// TIA Portal project "ABB_umrichter_Profinet" (V14)

(* hardware
DEVICE "S7-1200-Station_1"  S7-1200 Station
   slot 0: "Baugruppenträger_0"  S7-1200 Rack  Rack  V1.0
   slot 1: "PLC_1"  CPU 1214C DC/DC/DC  6ES7 214-1AG40-0XB0  V4.2
DEVICE "GSD-Geraet_1"  GSD.Device.PN
   slot 0: "Baugruppenträger"  Rack  V1.0
   slot 0: "FENA"  FENA-11  6438177287445  V3.2.0
      slot 0: "FENA-11"  FENA-11
      slot 1: "Interface"  Interface
         slot 1: "Port 1"  Port 1
   slot 1: "PPO Type 6_1"  PPO Type 6  V3.2.0
      slot 0: "PPO6 Data Object"  PPO6 Data Object
*)

// ===== PLC "PLC_1"  CPU 1214C DC/DC/DC =====

// folder: ABB_Datentypen

TYPE "ABB"
TITLE = ABB DRIVE CONTROL INPUT AND OUT FALGS
VERSION : 0.1
// Know_How_Protect
   STRUCT
      PPO_TYPE : "PPO_TYPE";
      ADAPTER_TYPE : "ADAPTER_TYPE";
      DRIVER_TYPE : "DRIVER_TYPE";
      DPV_MODE : "DPV_MODE";   // FALSE = DP-V0 ; TRUE = DP-V1
      SWITCH_ON : Bool;   // TRUE = switch on(power on);FALSE = switch off; start power on state machine
      START : Bool;   // TRUE = start enable modulation; FALSE = stop along currently activ stop ramp
      EMCY_STOP : Bool;   // Low active; emergency stop to drive: FALSE = stop by ramp TRUE = no stop
      COAST_STOP : Bool;   // TRUE = coast stop FALSE = normal operation eneble
      EXT_CTRL : Bool;   // External control place 2 EXT2
      RESET : Bool;   // Fault acknowled
      SPEED_REF : Int;   // Speed reference value: -20000...20000
      DONE : Bool;   // Execution finished when output DONE=TRUE
      ERR : Bool;   // Error occured during execution when output ERR=TRUE
      STOPPED : Bool;   // Drive stopped, not ready 0=ready
      RUNNING : Bool;   // Drive is modulating - following reference
      FAULT : Bool;   // Drive has a fault
      WARN : Bool;   // Drive has a warning
      EXT_RUN_ENABLE : Bool;   // External run enable singal received -> must be set to run
      LOACAL_CONTROL : Bool;   // Drive control location LOCAL
      EXT_CTRL_LOC : Bool;   // External control location EXT2 selected
      ERNO : Int;   // ErrorCode; see online help SFC14 or SFC15
      ACT_SPEED : Int;   // Speed actual value: -20000...20000
      MSW : Word;   // Main Status Word
      MCW : Word;   // Actual Main Control Word
      PARA_READ : Bool;   // Read parameter value
      PARA_WRITE : Bool;   // Write parameter value
      PARA_NUM : DInt;   // Parameter number: 3 digits = group, 2 digits = index; e.g Par 20.06 = 2006
      PARA_VALUE_IN : DInt;   // Write parameter value
      PARA_DONE : Bool;   // Pulse execution finished
      PARA_ERR : Bool;   // Error occured
      PARA_BUSY : Bool;   // Function block busy
      PARA_ERNO : Word;   // Error ID see FPBA or RBPA manual
      PARA_NUM_OUT : DInt;   // Parameter number: 3 digits = group, 2 digits = index; e.g Par 20.06 = 2006
      PARA_VALUE_OUT : DInt;   // Readed parameter value
      PZD3_OUT : Int;   // Write PZD3 value to drive
      PZD4_OUT : Int;   // Write PZD4 value to drive
      PZD5_OUT : Int;   // Write PZD5 value to drive
      PZD6_OUT : Int;   // Write PZD6 value to drive
      PZD7_OUT : Int;   // Write PZD7 value to drive
      PZD8_OUT : Int;   // Write PZD8 value to drive
      PZD9_OUT : Int;   // Write PZD9 value to drive
      PZD10_OUT : Int;   // Write PZD10 value to drive
      PZD2_SCALED : Real;   // PZD2 scaled value
      PZD3_SCALED : Real;   // PZD3 scaled value
      PZD4_SCALED : Real;   // PZD4 scaled value
      PZD5_SCALED : Real;   // PZD5 scaled value
      PZD6_SCALED : Real;   // PZD6 scaled value
      PZD7_SCALED : Real;   // PZD7 scaled value
      PZD8_SCALED : Real;   // PZD8 scaled value
      PZD9_SCALED : Real;   // PZD9 scaled value
      PZD10_SCALED : Real;   // PZD10 scaled value
   END_STRUCT;
END_TYPE

// folder: ABB_Datentypen/SUBTYPE

TYPE "PPO_TYPE"
   STRUCT
      PPP_TYPE1 : Int := 1;
      PPP_TYPE2 : Int := 2;
      PPP_TYPE3 : Int := 3;
      PPP_TYPE4 : Int := 4;
      PPP_TYPE5 : Int := 5;
      PPP_TYPE6 : Int := 6;
      PPP_TYPE7 : Int := 7;
   END_STRUCT;
END_TYPE

TYPE "DRIVER_TYPE"
   STRUCT
      ACS800 : Int := 1;
      ACSM1 : Int := 2;
      ACS350 : Int := 3;
      ACS355 : Int := 4;
      ACS550 : Int := 5;
      ACS850 : Int := 6;
      ACS880 : Int := 7;
      ACS580 : Int := 8;
      ACS380 : Int := 9;
   END_STRUCT;
END_TYPE

TYPE "ADAPTER_TYPE"
   STRUCT
      "FPBA/FENA" : Int := 1;
      "RPBA/RETA" : Int := 2;
   END_STRUCT;
END_TYPE

TYPE "DPV_MODE"
   STRUCT
      DP_V0 : Bool;
      "DP_V1/Profinet" : Bool := true;
   END_STRUCT;
END_TYPE

// folder: (top level)

DATA_BLOCK "GVL"   // DB2
{ S7_Optimized_Access := 'TRUE' }
VERSION : 0.1
   VAR
      Drive_Param : "ABB";
   END_VAR
BEGIN
   // Drive_Param.SWITCH_ON : FALSE=Drive control switched off, TRUE=Drive control switched on. After an EMERGENCY STOP a new rising edge of SWITCH_ON is needed before next start. SWITCH_ON also needs to be active (TRUE) for resetting drive faults.
   // Drive_Param.START : FALSE=Ramp stop with deceleration time according to drive parameter, TRUE=Start. Drive start via fieldbus requires parameter setting in the drive.
   // Drive_Param.EMCY_STOP : FALSE=Emergency stop according to emergency stop deceleration time set in drive parameter, TRUE=Normal operation.
   // Drive_Param.COAST_STOP : FALSE=Normal operation, TRUE=Coast stop (drive releases control of the motor).
   // Drive_Param.EXT_CTRL : Selection of external control location EXT2. FALSE=EXT1, TRUE=EXT2. Shifting to EXT2 via fieldbus requires parameter setting in the drive.
   // Drive_Param.DPV_MODE : FALSE=DP-V01, TRUE=DP-V12 (or PROFINET).
   // Drive_Param.RESET : FALSE=No operation, TRUE =Reset drive fault.
   // Drive_Param.SPEED_REF : Speed reference value: -20000 to 20000. See chapter “Drive configuration” for scaling. Setting speed reference via fieldbus requires parameter setting in the drive.
   // Drive_Param.DONE : FALSE=Block execution not finished, TRUE=Block execution finished.
   // Drive_Param.ERR : FALSE=No error, TRUE=Error occurred during block execution.
   // Drive_Param.STOPPED : FALSE=Drive is not stopped, TRUE=Drive is stopped.
   // Drive_Param.RUNNING : FALSE=Drive is not running, TRUE=Drive is running and following the speed reference value.
   // Drive_Param.FAULT : FALSE=No drive fault active, TRUE=Drive fault active.
   // Drive_Param.WARN : FALSE=No drive warning active, TRUE=Drive warning active.FALSE=No drive warning active, TRUE=Drive warning active.
   // Drive_Param.EXT_RUN_ENABLE : FALSE=No external run enable signal received in the drive, TRUE=External run enable signal received in the drive.
   // Drive_Param.LOACAL_CONTROL : FALSE=Remote control (normal mode), TRUE=Local control (e.g. drive control panel or pc tool in local mode)
   // Drive_Param.EXT_CTRL_LOC : Actual control place, FALSE=EXT1, TRUE=EXT2.
   // Drive_Param.ERNO : Error code when ERR=TRUE, see SIMATIC online help for SFC14 or SFC15.
   // Drive_Param.ACT_SPEED : Drive actual speed: -20000 to 20000. See chapter “Drive configuration” for scaling.
   // Drive_Param.MSW : Drive main status word. See actual fieldbus adapter manual for detailed description.
   // Drive_Param.MCW : Drive main control word. See actual fieldbus adapter manual for detailed description.
   // Drive_Param.PARA_READ : Read the parameter value 0 -> 1 (executed on positive edge).
   // Drive_Param.PARA_WRITE : Write the parameter value 0 -> 1 (executed on positive edge).
   // Drive_Param.PARA_NUM : Read/written parameter: 3 numbers = group, 2 numbers =
   // Drive_Param.PARA_VALUE_IN : Parameter value to be written.
   // Drive_Param.PARA_DONE : FALSE=Block execution not finished, TRUE=Block execution finished.
   // Drive_Param.PARA_ERR : FALSE=No error, TRUE=Error occurred during block execution.
   // Drive_Param.PARA_BUSY : FALSE=No operation active, TRUE=Operation active.
   // Drive_Param.PARA_ERNO : Error code when ERR=TRUE.
   // Drive_Param.PARA_NUM_OUT : Handled parameter number: 3 numbers = group, 2 numbers = index; for example, Par 20.06 = 2006.
   // Drive_Param.PARA_VALUE_OUT : Read parameter value.
   // Drive_Param.PZD3_OUT : Write PZD3 value to the drive
   // Drive_Param.PZD4_OUT : Write PZD4 value to the drive
   // Drive_Param.PZD5_OUT : Write PZD5 value to the drive
   // Drive_Param.PZD6_OUT : Write PZD6 value to the drive
   // Drive_Param.PZD7_OUT : Write PZD7 value to the drive
   // Drive_Param.PZD8_OUT : Write PZD8 value to the drive
   // Drive_Param.PZD9_OUT : Write PZD9 value to the drive
   // Drive_Param.PZD10_OUT : Write PZD10 value to the drive
   // Drive_Param.PZD2_SCALED : Read PZD2 (actual speed / ACT) value from the drive, the default
   // Drive_Param.PZD3_SCALED : Read PZD3 value from the drive, the default scaling value is 1 = no
   // Drive_Param.PZD4_SCALED : Read PZD4 value from the drive, the default scaling value is 1 = no
   // Drive_Param.PZD5_SCALED : Read PZD5 value from the drive, the default scaling value is 1 = no
   // Drive_Param.PZD6_SCALED : Read PZD6 value from the drive, the default scaling value is 1 = no
   // Drive_Param.PZD7_SCALED : Read PZD7 value from the drive, the default scaling value is 1 = no
   // Drive_Param.PZD8_SCALED : Read PZD8 value from the drive, the default scaling value is 1 = no
   // Drive_Param.PZD9_SCALED : Read PZD9 value from the drive, the default scaling value is 1 = no
   // Drive_Param.PZD10_SCALED : Read PZD10 value from the drive, the default scaling value is 1 = no
   // Drive_Param.PPO_TYPE : The PPO type. 1, 2, 3, 4, 5 or 6; 0 = not allowed.
   // Drive_Param.ADAPTER_TYPE : PROFIBUS module type: FPBA-01 PROFIBUS DP module connected in the drive. 1=FPBA (or FENA), 2=RPBA (or RETA).
   // Drive_Param.DRIVER_TYPE : Drive type: ACS800=1, ACSM1=2, ACS350=3, ACS355=4, ACS550=5, ACS850=6, ACS880=7, ACS580=8, ACS380=9.
END_DATA_BLOCK

// folder: ABB_Umrichter

DATA_BLOCK "ABB_Umrichter_DB"   // DB5
{ S7_Optimized_Access := 'TRUE' }
VERSION : 0.1
// stored: InstanceOfName ABB_Umrichter
"ABB_Umrichter"
BEGIN
END_DATA_BLOCK

// folder: ABB_Umrichter/DLL

DATA_BLOCK "ABB_DRIVE_CONTROL_DB"   // DB1
{ S7_Optimized_Access := 'FALSE' }
AUTHOR : ABB
FAMILY : DRIVES
NAME : ABB
VERSION : 1.2
// stored: InstanceOfName ABB_DRIVE_CONTROL
"ABB_DRIVE_CONTROL"
BEGIN
END_DATA_BLOCK

DATA_BLOCK "ACS_DRIVE_PARA_DB"   // DB3
{ S7_Optimized_Access := 'FALSE' }
AUTHOR : ABB
FAMILY : DRIVES
NAME : ABB
VERSION : 1.2
// stored: InstanceOfName ACS_DRIVE_PARA
"ACS_DRIVE_PARA"
BEGIN
END_DATA_BLOCK

DATA_BLOCK "ACS_DRIVE_PZD_DB"   // DB4
{ S7_Optimized_Access := 'FALSE' }
AUTHOR : ABB
FAMILY : DRIVES
NAME : ABB
VERSION : 1.2
// stored: InstanceOfName ACS_DRIVE_PZD
"ACS_DRIVE_PZD"
BEGIN
END_DATA_BLOCK

// folder: (top level)

ORGANIZATION_BLOCK "Main"   // OB1, LAD, ProgramCycle
TITLE = "Main Program Sweep (Cycle)"
{ S7_Optimized_Access := 'TRUE' }
VERSION : 0.1
   VAR_INPUT
      Initial_Call : Bool;   // Initial call of this OB
      Remanence : Bool;   // =True, if remanent data are available
   END_VAR
BEGIN

REGION Network 1
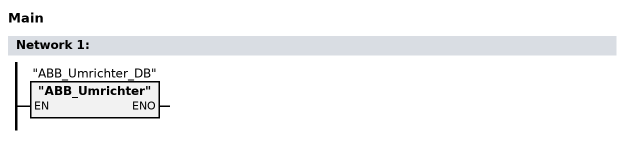
   RUNG wire#powerrail
      "ABB_Umrichter_DB"()
   END_RUNG
   // the same network as SCL:
   "ABB_Umrichter_DB"();   // "ABB_Umrichter"
END_REGION
END_ORGANIZATION_BLOCK

// folder: ABB_Umrichter

FUNCTION_BLOCK "ABB_Umrichter"   // FB1, LAD
{ S7_Optimized_Access := 'TRUE' }
VERSION : 0.1
BEGIN

REGION Network 1
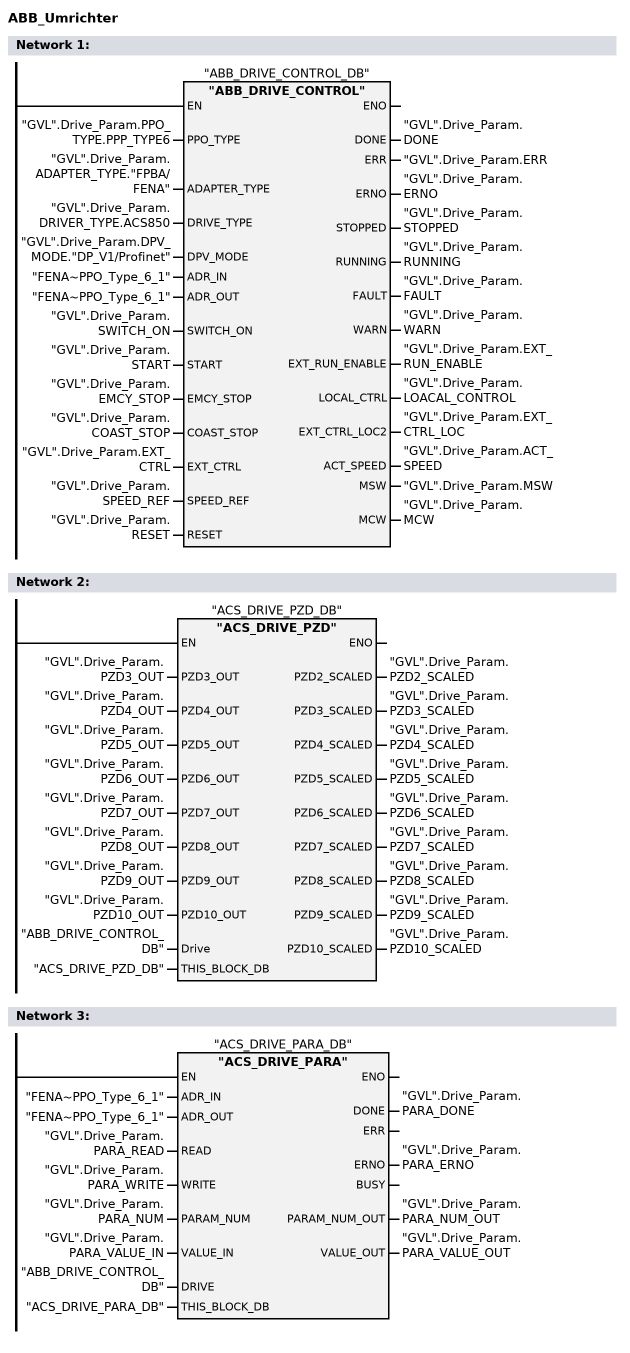
   RUNG wire#powerrail
      "ABB_DRIVE_CONTROL_DB"(PPO_TYPE := "GVL".Drive_Param.PPO_TYPE.PPP_TYPE6, ADAPTER_TYPE := "GVL".Drive_Param.ADAPTER_TYPE."FPBA/FENA", DRIVE_TYPE := "GVL".Drive_Param.DRIVER_TYPE.ACS850, DPV_MODE := "GVL".Drive_Param.DPV_MODE."DP_V1/Profinet", ADR_IN := "FENA~PPO_Type_6_1", ADR_OUT := "FENA~PPO_Type_6_1", SWITCH_ON := "GVL".Drive_Param.SWITCH_ON, START := "GVL".Drive_Param.START, EMCY_STOP := "GVL".Drive_Param.EMCY_STOP, COAST_STOP := "GVL".Drive_Param.COAST_STOP, EXT_CTRL := "GVL".Drive_Param.EXT_CTRL, SPEED_REF := "GVL".Drive_Param.SPEED_REF, RESET := "GVL".Drive_Param.RESET, DONE => "GVL".Drive_Param.DONE, ERR => "GVL".Drive_Param.ERR, ERNO => "GVL".Drive_Param.ERNO, STOPPED => "GVL".Drive_Param.STOPPED, RUNNING => "GVL".Drive_Param.RUNNING, FAULT => "GVL".Drive_Param.FAULT, WARN => "GVL".Drive_Param.WARN, EXT_RUN_ENABLE => "GVL".Drive_Param.EXT_RUN_ENABLE, LOCAL_CTRL => "GVL".Drive_Param.LOACAL_CONTROL, EXT_CTRL_LOC2 => "GVL".Drive_Param.EXT_CTRL_LOC, ACT_SPEED => "GVL".Drive_Param.ACT_SPEED, MSW => "GVL".Drive_Param.MSW, MCW => "GVL".Drive_Param.MCW)
   END_RUNG
   // the same network as SCL:
   "ABB_DRIVE_CONTROL_DB"(PPO_TYPE := "GVL".Drive_Param.PPO_TYPE.PPP_TYPE6,   // "ABB_DRIVE_CONTROL"
                          ADAPTER_TYPE := "GVL".Drive_Param.ADAPTER_TYPE."FPBA/FENA",
                          DRIVE_TYPE := "GVL".Drive_Param.DRIVER_TYPE.ACS850,
                          DPV_MODE := "GVL".Drive_Param.DPV_MODE."DP_V1/Profinet",
                          ADR_IN := "FENA~PPO_Type_6_1",
                          ADR_OUT := "FENA~PPO_Type_6_1",
                          SWITCH_ON := "GVL".Drive_Param.SWITCH_ON,
                          START := "GVL".Drive_Param.START,
                          EMCY_STOP := "GVL".Drive_Param.EMCY_STOP,
                          COAST_STOP := "GVL".Drive_Param.COAST_STOP,
                          EXT_CTRL := "GVL".Drive_Param.EXT_CTRL,
                          SPEED_REF := "GVL".Drive_Param.SPEED_REF,
                          RESET := "GVL".Drive_Param.RESET,
                          DONE => "GVL".Drive_Param.DONE,
                          ERR => "GVL".Drive_Param.ERR,
                          ERNO => "GVL".Drive_Param.ERNO,
                          STOPPED => "GVL".Drive_Param.STOPPED,
                          RUNNING => "GVL".Drive_Param.RUNNING,
                          FAULT => "GVL".Drive_Param.FAULT,
                          WARN => "GVL".Drive_Param.WARN,
                          EXT_RUN_ENABLE => "GVL".Drive_Param.EXT_RUN_ENABLE,
                          LOCAL_CTRL => "GVL".Drive_Param.LOACAL_CONTROL,
                          EXT_CTRL_LOC2 => "GVL".Drive_Param.EXT_CTRL_LOC,
                          ACT_SPEED => "GVL".Drive_Param.ACT_SPEED,
                          MSW => "GVL".Drive_Param.MSW,
                          MCW => "GVL".Drive_Param.MCW);
END_REGION

REGION Network 2
   RUNG wire#powerrail
      "ACS_DRIVE_PZD_DB"(PZD3_OUT := "GVL".Drive_Param.PZD3_OUT, PZD4_OUT := "GVL".Drive_Param.PZD4_OUT, PZD5_OUT := "GVL".Drive_Param.PZD5_OUT, PZD6_OUT := "GVL".Drive_Param.PZD6_OUT, PZD7_OUT := "GVL".Drive_Param.PZD7_OUT, PZD8_OUT := "GVL".Drive_Param.PZD8_OUT, PZD9_OUT := "GVL".Drive_Param.PZD9_OUT, PZD10_OUT := "GVL".Drive_Param.PZD10_OUT, Drive := "ABB_DRIVE_CONTROL_DB", THIS_BLOCK_DB := "ACS_DRIVE_PZD_DB", PZD2_SCALED => "GVL".Drive_Param.PZD2_SCALED, PZD3_SCALED => "GVL".Drive_Param.PZD3_SCALED, PZD4_SCALED => "GVL".Drive_Param.PZD4_SCALED, PZD5_SCALED => "GVL".Drive_Param.PZD5_SCALED, PZD6_SCALED => "GVL".Drive_Param.PZD6_SCALED, PZD7_SCALED => "GVL".Drive_Param.PZD7_SCALED, PZD8_SCALED => "GVL".Drive_Param.PZD8_SCALED, PZD9_SCALED => "GVL".Drive_Param.PZD9_SCALED, PZD10_SCALED => "GVL".Drive_Param.PZD10_SCALED)
   END_RUNG
   // the same network as SCL:
   "ACS_DRIVE_PZD_DB"(PZD3_OUT := "GVL".Drive_Param.PZD3_OUT,   // "ACS_DRIVE_PZD"
                      PZD4_OUT := "GVL".Drive_Param.PZD4_OUT,
                      PZD5_OUT := "GVL".Drive_Param.PZD5_OUT,
                      PZD6_OUT := "GVL".Drive_Param.PZD6_OUT,
                      PZD7_OUT := "GVL".Drive_Param.PZD7_OUT,
                      PZD8_OUT := "GVL".Drive_Param.PZD8_OUT,
                      PZD9_OUT := "GVL".Drive_Param.PZD9_OUT,
                      PZD10_OUT := "GVL".Drive_Param.PZD10_OUT,
                      Drive := "ABB_DRIVE_CONTROL_DB",
                      THIS_BLOCK_DB := "ACS_DRIVE_PZD_DB",
                      PZD2_SCALED => "GVL".Drive_Param.PZD2_SCALED,
                      PZD3_SCALED => "GVL".Drive_Param.PZD3_SCALED,
                      PZD4_SCALED => "GVL".Drive_Param.PZD4_SCALED,
                      PZD5_SCALED => "GVL".Drive_Param.PZD5_SCALED,
                      PZD6_SCALED => "GVL".Drive_Param.PZD6_SCALED,
                      PZD7_SCALED => "GVL".Drive_Param.PZD7_SCALED,
                      PZD8_SCALED => "GVL".Drive_Param.PZD8_SCALED,
                      PZD9_SCALED => "GVL".Drive_Param.PZD9_SCALED,
                      PZD10_SCALED => "GVL".Drive_Param.PZD10_SCALED);
END_REGION

REGION Network 3
   RUNG wire#powerrail
      "ACS_DRIVE_PARA_DB"(ADR_IN := "FENA~PPO_Type_6_1", ADR_OUT := "FENA~PPO_Type_6_1", READ := "GVL".Drive_Param.PARA_READ, WRITE := "GVL".Drive_Param.PARA_WRITE, PARAM_NUM := "GVL".Drive_Param.PARA_NUM, VALUE_IN := "GVL".Drive_Param.PARA_VALUE_IN, DRIVE := "ABB_DRIVE_CONTROL_DB", THIS_BLOCK_DB := "ACS_DRIVE_PARA_DB", DONE => "GVL".Drive_Param.PARA_DONE, ERR =>, ERNO => "GVL".Drive_Param.PARA_ERNO, BUSY =>, PARAM_NUM_OUT => "GVL".Drive_Param.PARA_NUM_OUT, VALUE_OUT => "GVL".Drive_Param.PARA_VALUE_OUT)
   END_RUNG
   // the same network as SCL:
   "ACS_DRIVE_PARA_DB"(ADR_IN := "FENA~PPO_Type_6_1",   // "ACS_DRIVE_PARA"
                       ADR_OUT := "FENA~PPO_Type_6_1",
                       READ := "GVL".Drive_Param.PARA_READ,
                       WRITE := "GVL".Drive_Param.PARA_WRITE,
                       PARAM_NUM := "GVL".Drive_Param.PARA_NUM,
                       VALUE_IN := "GVL".Drive_Param.PARA_VALUE_IN,
                       DRIVE := "ABB_DRIVE_CONTROL_DB",
                       THIS_BLOCK_DB := "ACS_DRIVE_PARA_DB",
                       DONE => "GVL".Drive_Param.PARA_DONE,
                       ERNO => "GVL".Drive_Param.PARA_ERNO,
                       PARAM_NUM_OUT => "GVL".Drive_Param.PARA_NUM_OUT,
                       VALUE_OUT => "GVL".Drive_Param.PARA_VALUE_OUT);
END_REGION
END_FUNCTION_BLOCK

// folder: ABB_Umrichter/DLL

FUNCTION_BLOCK "ABB_DRIVE_CONTROL"   // FB500, LAD
TITLE = ABB_DRIVE_CONTROL_FB
{ S7_Optimized_Access := 'FALSE' }
AUTHOR : ABB
FAMILY : DRIVES
NAME : ABB
VERSION : 1.2
   VAR_INPUT
      PPO_TYPE : Int;   // PPO-Type: 1,2,3,4,5 or 6; 0 = no fuction
      ADAPTER_TYPE : Int;   // AdapterType:FPBA=1,RPBA=2,FENA=3
      DRIVE_TYPE : Int;   // DriveType: ACS800=1,ACSM1=2,ACS350=3,ACS355=4,ACS550=5,ACS850=6,ACS880=7,ACS580=8,ACS380=9
      DPV_MODE : Bool;   // FALSE = DP-V0 ; TRUE = DP-V1
      ADR_IN : Hw_Io;   // Address of first input byte
      ADR_OUT : Hw_Io;   // Address of first output byte
      SWITCH_ON : Bool;   // TRUE = switch on(power on);FALSE = switch off; start power on state machine
      START : Bool;   // TRUE = start enable modulation; FALSE = stop along currently activ stop ramp
      EMCY_STOP : Bool;   // Low active; emergency stop to drive: FALSE = stop by ramp TRUE = no stop
      COAST_STOP : Bool;   // TRUE = coast stop FALSE = normal operation eneble
      EXT_CTRL : Bool;   // External control place 2 EXT2
      SPEED_REF : Int;   // Speed reference value: -20000...20000
   END_VAR
   VAR_OUTPUT
      DONE : Bool;   // Execution finished when output DONE=TRUE
      ERR : Bool;   // Error occured during execution when output ERR=TRUE
      ERNO : Int;   // ErrorCode; see online help SFC14 or SFC15
      STOPPED : Bool;   // The drive has been stopped
      RUNNING : Bool;   // Drive is modulating - following reference
      FAULT : Bool;   // Drive has a fault
      WARN : Bool;   // Drive has a warning
      EXT_RUN_ENABLE : Bool;   // External run enable singal received -> must be set to run
      LOCAL_CTRL : Bool;   // Drive control location LOCAL
      EXT_CTRL_LOC2 : Bool;   // External control location EXT2 selected
      ACT_SPEED : Int;   // Speed actual value: -20000...20000
      MSW : Word;   // Main Status Word
      MCW : Word;   // Actual Main Control Word
   END_VAR
   VAR_IN_OUT
      RESET : Bool;   // Fault acknowled
   END_VAR
   VAR
      Input : Struct
         PPO1 : Struct
            SW : Struct
               AT_SET_POINT : Bool;   // Speed within setpoints
               REMONTE : Bool;   // Profibus control allowed
               ABOVE_LIMIT : Bool;   // Speed / frequency across borders
               EXT_CTRL_LOC : Bool;   // 0=EXT1 1=EXT2 selected
               EXT_RUN_ENABLE : Bool;   // Injury Prevention
               MSV13 : Bool;   // Not in Use
               MSV14 : Bool;   // Not in Use
               COOM_FAULT : Bool;   // Communication Fault Profibus Module CH0
               RDY_ON : Bool;   // Startup finished
               RDY_RUN : Bool;   // Action Completed
               RDY_REF : Bool;   // In Progress
               TRIPPED : Bool;   // Interference
               OFF2_STATE : Bool;   // Freedom freely in the wheels
               OFF3_STATE : Bool;   // Stop as fast as possible
               ON_INHIB : Bool;   // Startup blocked
               ALARM : Bool;   // Alarm
            END_STRUCT;
            Act_Speed : Int;   // Speed
         END_STRUCT;
         PPO2 : Struct
            SW : Struct
               AT_SET_POINT : Bool;   // Speed within setpoints
               REMONTE : Bool;   // Profibus control allowed
               ABOVE_LIMIT : Bool;   // Speed / frequency across borders
               EXT_CTRL_LOC : Bool;   // 0=EXT1 1=EXT2 selected
               EXT_RUN_ENABLE : Bool;   // Injury Prevention
               MSV13 : Bool;   // Not in Use
               MSV14 : Bool;   // Not in Use
               COOM_FAULT : Bool;   // Communication Fault Profibus Module CH0
               RDY_ON : Bool;   // Startup finished
               RDY_RUN : Bool;   // Action Completed
               RDY_REF : Bool;   // In Progress
               TRIPPED : Bool;   // Interference
               OFF2_STATE : Bool;   // Freedom freely in the wheels
               OFF3_STATE : Bool;   // Stop as fast as possible
               ON_INHIB : Bool;   // Startup blocked
               ALARM : Bool;   // Alarm
            END_STRUCT;
            Act_Speed : Int;   // Speed
            PZD_3 : Int;
            PZD_4 : Int;
            PZD_5 : Int;
            PZD_6 : Int;
         END_STRUCT;
         PPO3 : Struct
            SW : Struct
               AT_SET_POINT : Bool;   // Speed within setpoints
               REMONTE : Bool;   // Profibus control allowed
               ABOVE_LIMIT : Bool;   // Speed / frequency across borders
               EXT_CTRL_LOC : Bool;   // 0=EXT1 1=EXT2 selected
               EXT_RUN_ENABLE : Bool;   // Injury Prevention
               MSV13 : Bool;   // Not in Use
               MSV14 : Bool;   // Not in Use
               COOM_FAULT : Bool;   // Communication Fault Profibus Module CH0
               RDY_ON : Bool;   // Startup finished
               RDY_RUN : Bool;   // Action Completed
               RDY_REF : Bool;   // In Progress
               TRIPPED : Bool;   // Interference
               OFF2_STATE : Bool;   // Freedom freely in the wheels
               OFF3_STATE : Bool;   // Stop as fast as possible
               ON_INHIB : Bool;   // Startup blocked
               ALARM : Bool;   // Alarm
            END_STRUCT;
            Act_Speed : Int;   // Speed
         END_STRUCT;
         PPO4 : Struct
            SW : Struct
               AT_SET_POINT : Bool;   // Speed within setpoints
               REMONTE : Bool;   // Profibus control allowed
               ABOVE_LIMIT : Bool;   // Speed / frequency across borders
               EXT_CTRL_LOC : Bool;   // 0=EXT1 1=EXT2 selected
               EXT_RUN_ENABLE : Bool;   // Injury Prevention
               MSV13 : Bool;   // Not in Use
               MSV14 : Bool;   // Not in Use
               COOM_FAULT : Bool;   // Communication Fault Profibus Module CH0
               RDY_ON : Bool;   // Startup finished
               RDY_RUN : Bool;   // Action Completed
               RDY_REF : Bool;   // In Progress
               TRIPPED : Bool;   // Interference
               OFF2_STATE : Bool;   // Freedom freely in the wheels
               OFF3_STATE : Bool;   // Stop as fast as possible
               ON_INHIB : Bool;   // Startup blocked
               ALARM : Bool;   // Alarm
            END_STRUCT;
            Act_Speed : Int;   // Speed
            PZD_3 : Int;
            PZD_4 : Int;
            PZD_5 : Int;
            PZD_6 : Int;
         END_STRUCT;
         PPO5 : Struct
            SW : Struct
               AT_SET_POINT : Bool;   // Speed within setpoints
               REMONTE : Bool;   // Profibus control allowed
               ABOVE_LIMIT : Bool;   // Speed / frequency across borders
               EXT_CTRL_LOC : Bool;   // 0=EXT1 1=EXT2 selected
               EXT_RUN_ENABLE : Bool;   // Injury Prevention
               MSV13 : Bool;   // Not in Use
               MSV14 : Bool;   // Not in Use
               COOM_FAULT : Bool;   // Communication Fault Profibus Module CH0
               RDY_ON : Bool;   // Startup finished
               RDY_RUN : Bool;   // Action Completed
               RDY_REF : Bool;   // In Progress
               TRIPPED : Bool;   // Interference
               OFF2_STATE : Bool;   // Freedom freely in the wheels
               OFF3_STATE : Bool;   // Stop as fast as possible
               ON_INHIB : Bool;   // Startup blocked
               ALARM : Bool;   // Alarm
            END_STRUCT;
            Act_Speed : Int;   // Speed
            PZD_3 : Int;
            PZD_4 : Int;
            PZD_5 : Int;
            PZD_6 : Int;
            PZD_7 : Int;
            PZD_8 : Int;
            PZD_9 : Int;
            PZD_10 : Int;
         END_STRUCT;
         PPO6 : Struct
            SW : Struct
               AT_SET_POINT : Bool;   // Speed within setpoints
               REMONTE : Bool;   // Profibus control allowed
               ABOVE_LIMIT : Bool;   // Speed / frequency across borders
               EXT_CTRL_LOC : Bool;   // 0=EXT1 1=EXT2 selected
               EXT_RUN_ENABLE : Bool;   // Injury Prevention
               MSV13 : Bool;   // Not in Use
               MSV14 : Bool;   // Not in Use
               COOM_FAULT : Bool;   // Communication Fault Profibus Module CH0
               RDY_ON : Bool;   // Startup finished
               RDY_RUN : Bool;   // Action Completed
               RDY_REF : Bool;   // In Progress
               TRIPPED : Bool;   // Interference
               OFF2_STATE : Bool;   // Freedom freely in the wheels
               OFF3_STATE : Bool;   // Stop as fast as possible
               ON_INHIB : Bool;   // Startup blocked
               ALARM : Bool;   // Alarm
            END_STRUCT;
            Act_Speed : Int;   // Speed
            PZD_3 : Int;
            PZD_4 : Int;
            PZD_5 : Int;
            PZD_6 : Int;
            PZD_7 : Int;
            PZD_8 : Int;
            PZD_9 : Int;
            PZD_10 : Int;
         END_STRUCT;
         ACT : Struct
            SW : Struct
               AT_SET_POINT : Bool;   // Speed within setpoints
               REMONTE : Bool;   // Profibus control allowed
               ABOVE_LIMIT : Bool;   // Speed / frequency across borders
               EXT_CTRL_LOC : Bool;   // 0=EXT1 1=EXT2 selected
               EXT_RUN_ENABLE : Bool;   // Injury Prevention
               MSV13 : Bool;   // Not in Use
               MSV14 : Bool;   // Not in Use
               COOM_FAULT : Bool;   // Communication Fault Profibus Module CH0
               RDY_ON : Bool;   // Startup finished
               RDY_RUN : Bool;   // Action Completed
               RDY_REF : Bool;   // In Progress
               TRIPPED : Bool;   // Interference
               OFF2_STATE : Bool;   // Freedom freely in the wheels
               OFF3_STATE : Bool;   // Stop as fast as possible
               ON_INHIB : Bool;   // Startup blocked
               ALARM : Bool;   // Alarm
            END_STRUCT;
            Act_Speed : Int;   // Speed
         END_STRUCT;
      END_STRUCT;
      Output : Struct
         PPO1 : Struct
            CW : Struct
               INCHING_1 : Bool;   // Standard Speed for instruction 1
               INCHING_2 : Bool;   // Standard Speed for instruction 2
               REMONTE_CMD : Bool;   // Profibus control for use
               EXT_CTRL_LOC : Bool;   // 0=EXT1 1=EXT2 selected
               RESERVE_2 : Bool;   // Not in Use
               RESERVE_3 : Bool;   // Not in Use
               RESERVE_4 : Bool;   // Not in Use
               RESERVE_5 : Bool;   // Not in Use
               OFF1 : Bool;   // Start up to readiness
               OFF2 : Bool;   // Free wheel stops
               OFF3 : Bool;   // Emergency stop stop
               INHIBIT_OPREATION : Bool;   // Go to control
               RAMP_OUT_ZERO : Bool;   // Control release
               RAMP_HOLD : Bool;   // Acceleration allowed
               RAMP_IN_ZERO : Bool;   // Speed instruction to zero
               RESET : Bool;   // Fault Reset
            END_STRUCT;
            RefSpeed : Int;
         END_STRUCT;
         PPO2 : Struct
            CW : Struct
               INCHING_1 : Bool;   // Standard Speed for instruction 1
               INCHING_2 : Bool;   // Standard Speed for instruction 2
               REMONTE_CMD : Bool;   // Profibus control for use
               EXT_CTRL_LOC : Bool;   // 0=EXT1 1=EXT2 selected
               RESERVE_2 : Bool;   // Not in Use
               RESERVE_3 : Bool;   // Not in Use
               RESERVE_4 : Bool;   // Not in Use
               RESERVE_5 : Bool;   // Not in Use
               OFF1 : Bool;   // Start up to readiness
               OFF2 : Bool;   // Free wheel stops
               OFF3 : Bool;   // Emergency stop stop
               INHIBIT_OPREATION : Bool;   // Go to control
               RAMP_OUT_ZERO : Bool;   // Control release
               RAMP_HOLD : Bool;   // Acceleration allowed
               RAMP_IN_ZERO : Bool;   // Speed instruction to zero
               RESET : Bool;   // Fault Reset
            END_STRUCT;
            RefSpeed : Int;
            PZD_3 : Int;
            PZD_4 : Int;
            PZD_5 : Int;
            PZD_6 : Int;
         END_STRUCT;
         PPO3 : Struct
            CW : Struct
               INCHING_1 : Bool;   // Standard Speed for instruction 1
               INCHING_2 : Bool;   // Standard Speed for instruction 2
               REMONTE_CMD : Bool;   // Profibus control for use
               EXT_CTRL_LOC : Bool;   // 0=EXT1 1=EXT2 selected
               RESERVE_2 : Bool;   // Not in Use
               RESERVE_3 : Bool;   // Not in Use
               RESERVE_4 : Bool;   // Not in Use
               RESERVE_5 : Bool;   // Not in Use
               OFF1 : Bool;   // Start up to readiness
               OFF2 : Bool;   // Free wheel stops
               OFF3 : Bool;   // Emergency stop stop
               INHIBIT_OPREATION : Bool;   // Go to control
               RAMP_OUT_ZERO : Bool;   // Control release
               RAMP_HOLD : Bool;   // Acceleration allowed
               RAMP_IN_ZERO : Bool;   // Speed instruction to zero
               RESET : Bool;   // Fault Reset
            END_STRUCT;
            RefSpeed : Int;
         END_STRUCT;
         PPO4 : Struct
            CW : Struct
               INCHING_1 : Bool;   // Standard Speed for instruction 1
               INCHING_2 : Bool;   // Standard Speed for instruction 2
               REMONTE_CMD : Bool;   // Profibus control for use
               EXT_CTRL_LOC : Bool;   // 0=EXT1 1=EXT2 selected
               RESERVE_2 : Bool;   // Not in Use
               RESERVE_3 : Bool;   // Not in Use
               RESERVE_4 : Bool;   // Not in Use
               RESERVE_5 : Bool;   // Not in Use
               OFF1 : Bool;   // Start up to readiness
               OFF2 : Bool;   // Free wheel stops
               OFF3 : Bool;   // Emergency stop stop
               INHIBIT_OPREATION : Bool;   // Go to control
               RAMP_OUT_ZERO : Bool;   // Control release
               RAMP_HOLD : Bool;   // Acceleration allowed
               RAMP_IN_ZERO : Bool;   // Speed instruction to zero
               RESET : Bool;   // Fault Reset
            END_STRUCT;
            RefSpeed : Int;
            PZD_3 : Int;
            PZD_4 : Int;
            PZD_5 : Int;
            PZD_6 : Int;
         END_STRUCT;
         PPO5 : Struct
            CW : Struct
               INCHING_1 : Bool;   // Standard Speed for instruction 1
               INCHING_2 : Bool;   // Standard Speed for instruction 2
               REMONTE_CMD : Bool;   // Profibus control for use
               EXT_CTRL_LOC : Bool;   // 0=EXT1 1=EXT2 selected
               RESERVE_2 : Bool;   // Not in Use
               RESERVE_3 : Bool;   // Not in Use
               RESERVE_4 : Bool;   // Not in Use
               RESERVE_5 : Bool;   // Not in Use
               OFF1 : Bool;   // Start up to readiness
               OFF2 : Bool;   // Free wheel stops
               OFF3 : Bool;   // Emergency stop stop
               INHIBIT_OPREATION : Bool;   // Go to control
               RAMP_OUT_ZERO : Bool;   // Control release
               RAMP_HOLD : Bool;   // Acceleration allowed
               RAMP_IN_ZERO : Bool;   // Speed instruction to zero
               RESET : Bool;   // Fault Reset
            END_STRUCT;
            RefSpeed : Int;
            PZD_3 : Int;
            PZD_4 : Int;
            PZD_5 : Int;
            PZD_6 : Int;
            PZD_7 : Int;
            PZD_8 : Int;
            PZD_9 : Int;
            PZD_10 : Int;
         END_STRUCT;
         PPO6 : Struct
            CW : Struct
               INCHING_1 : Bool;   // Standard Speed for instruction 1
               INCHING_2 : Bool;   // Standard Speed for instruction 2
               REMONTE_CMD : Bool;   // Profibus control for use
               EXT_CTRL_LOC : Bool;   // 0=EXT1 1=EXT2 selected
               RESERVE_2 : Bool;   // Not in Use
               RESERVE_3 : Bool;   // Not in Use
               RESERVE_4 : Bool;   // Not in Use
               RESERVE_5 : Bool;   // Not in Use
               OFF1 : Bool;   // Start up to readiness
               OFF2 : Bool;   // Free wheel stops
               OFF3 : Bool;   // Emergency stop stop
               INHIBIT_OPREATION : Bool;   // Go to control
               RAMP_OUT_ZERO : Bool;   // Control release
               RAMP_HOLD : Bool;   // Acceleration allowed
               RAMP_IN_ZERO : Bool;   // Speed instruction to zero
               RESET : Bool;   // Fault Reset
            END_STRUCT;
            RefSpeed : Int;
            PZD_3 : Int;
            PZD_4 : Int;
            PZD_5 : Int;
            PZD_6 : Int;
            PZD_7 : Int;
            PZD_8 : Int;
            PZD_9 : Int;
            PZD_10 : Int;
         END_STRUCT;
         ACT : Struct
            CW : Struct
               INCHING_1 : Bool;   // Standard Speed for instruction 1
               INCHING_2 : Bool;   // Standard Speed for instruction 2
               REMONTE_CMD : Bool;   // Profibus control for use
               EXT_CTRL_LOC : Bool;   // 0=EXT1 1=EXT2 selected
               RESERVE_2 : Bool;   // Not in Use
               RESERVE_3 : Bool;   // Not in Use
               RESERVE_4 : Bool;   // Not in Use
               RESERVE_5 : Bool;   // Not in Use
               OFF1 : Bool;   // Start up to readiness
               OFF2 : Bool;   // Free wheel stops
               OFF3 : Bool;   // Emergency stop stop
               INHIBIT_OPREATION : Bool;   // Go to control
               RAMP_OUT_ZERO : Bool;   // Control release
               RAMP_HOLD : Bool;   // Acceleration allowed
               RAMP_IN_ZERO : Bool;   // Speed instruction to zero
               RESET : Bool;   // Fault Reset
            END_STRUCT;
            RefSpeed : Int;
         END_STRUCT;
      END_STRUCT;
      PARA_INTERNAL_DPV0 : Struct
         Done : Bool;
         Err : Bool;
         Busy : Bool;
         Read_FB : Bool;
         Write_FB : Bool;
         Time_out : Bool;
         Read_request : Bool;
         Write_Request : Bool;
         Parameter_access : Bool;
         Para_9 : Bool;
         Para_10 : Bool;
         Para_11 : Bool;
         Para_12 : Bool;
         Para_13 : Bool;
         Para_14 : Bool;
         Para_15 : Bool;
         Para_16 : Bool;
         Para_17 : Bool;
         Para_18 : Bool;
         Para_19 : Bool;
         Para_20 : Bool;
         Para_21 : Bool;
         Para_22 : Bool;
         Para_23 : Bool;
         Para_24 : Bool;
         Para_25 : Bool;
         Para_26 : Bool;
         Para_27 : Bool;
         Para_28 : Bool;
         Para_29 : Bool;
         Para_30 : Bool;
         PDV_MODE : Bool;   // DP-V0 = 0 (false) / DP-V1 = 1 (true)
         RESPONCE_LABEL : Int;
         PARA_NUM_OUT : Int;
         PARA_NUM_INDEX_OUT : Int;
         PARA_ERR_NRO : Word;
         PARA_VALUE_OUT : DInt;
         ADDRESS_IN : Word;
         ADDRESS_OUT : Word;
         Master_to_Slave : Struct
            ID : Word;   // Request Label bits 4-7 Parameter number bits 0-2
            IND : Word;   // Parameter number index bits 0-15
            VALUE : DWord;   // Parameter values
         END_STRUCT;
         Slave_to_Master : Struct
            ID : Word;   // Request Label bits 4-7 Parameter number bits 0-2
            IND : Word;   // Parameter number index bits 0-15
            VALUE : DWord;   // Parameter values
         END_STRUCT;
         PPO_TYPE : Int;   // PPO-Type: 1,2,3,4,5 or 6; 0 = no fuction
         ADAPTER_TYPE : Int;   // AdapterType:FPBA=1,RPBA=2,FENA=3
         DRIVE_TYPE : Int;   // DiveType: ACS800=1,ACSM1=2,ACS350=3,ACS355=4,ACS550=5,ACS850=6,ACS880=7
      END_STRUCT;
      PARA_INTERNAL_DPV1 : Struct
         Request : Struct
            Reference : Byte;
            ID : Byte;   // 1 read / 2 change
            Axis : Byte;
            NoOfParameters : Byte;
            Attribute : Byte;
            NoOfElements : Byte;
            ParameterIndex : Word;
            Subindex : Word;
            Format : Byte;
            NumberOfValues : Byte;
            Value : DWord;
         END_STRUCT;
         Responce : Struct
            Reference : Byte;
            ID : Byte;
            Axis : Byte;
            NoOfParametrs : Byte;
            Format : Byte;
            NoOfValues : Byte;
            Value : DWord;
         END_STRUCT;
         Request_DONE : Bool;
         Request_BUSY : Bool;
         Request_ERROR : Bool;
         Request_STATUS : DWord;
         Responce_VALID : Bool;
         Responce_BUSY : Bool;
         Responce_ERROR : Bool;
         Responce_STATUS : DWord;
         Responce_LEN : UInt;
      END_STRUCT;
      INTERNAL_PZD : Struct
         IN : Struct
            PZD2 : Int;
            PZD3 : Int;
            PZD4 : Int;
            PZD5 : Int;
            PZD6 : Int;
            PZD7 : Int;
            PZD8 : Int;
            PZD9 : Int;
            PZD10 : Int;
         END_STRUCT;
         OUT : Struct
            PZD3 : Int;
            PZD4 : Int;
            PZD5 : Int;
            PZD6 : Int;
            PZD7 : Int;
            PZD8 : Int;
            PZD9 : Int;
            PZD10 : Int;
         END_STRUCT;
         SCALED : Struct
            PZD2 : Real;
            PZD3 : Real;
            PZD4 : Real;
            PZD5 : Real;
            PZD6 : Real;
            PZD7 : Real;
            PZD8 : Real;
            PZD9 : Real;
            PZD10 : Real;
         END_STRUCT;
         SCALE : Struct
            PZD2_SCALE : Real;
            PZD3_SCALE : Real;
            PZD4_SCALE : Real;
            PZD5_SCALE : Real;
            PZD6_SCALE : Real;
            PZD7_SCALE : Real;
            PZD8_SCALE : Real;
            PZD9_SCALE : Real;
            PZD10_SCALE : Real;
         END_STRUCT;
      END_STRUCT;
      DPV1_WRITE : WRREC;
      DPV1_READ : WRREC;
      DP1_RESPONCE : RDREC;
      INPUT_ADDRESS : Word;
      OUTPUT_ADDRESS : Word;
      RET_VAL_INPUT : Int;
      RET_VAL_OUTPUT : Int;
      DONE_ON : Bool;
      ParameterErr : Bool;
      ERROR : Bool;
      READ_FAULT : Bool;
      SWITCH_ON_FP : Bool;
      POWER_STATE : Int;
      ALLWAYS_ON : Bool;
      ALLWAYS_OFF : Bool;
      POWER_ON : Bool;
      RESET_POWER_ON : Bool;
      PARA_TIME_OUT : TON_TIME;
      INTERNA_ERR : Int;
      POWER_RESET_FB : Bool;
      PARA_NUM : DInt;
      PARA_VALUE : DInt;
      PARA_INTERNAL_DPV1_16bit : Struct
         Request : Struct
            Reference : Byte;
            ID : Byte;   // 1 read / 2 change
            Axis : Byte;
            NoOfParameters : Byte;
            Attribute : Byte := B#16#10;
            NoOfElements : Byte;
            ParameterIndex : Word;
            Subindex : Word;
            Format : Byte;
            NumberOfValues : Byte;
            Value : Word;
         END_STRUCT;
         Responce : Struct
            Reference : Byte;
            ID : Byte;
            Axis : Byte;
            NoOfParametrs : Byte;
            Format : Byte;
            NoOfValues : Byte;
            Value : DWord;
         END_STRUCT;
         Request_DONE : Bool;
         Request_BUSY : Bool;
         Request_ERROR : Bool;
         Request_STATUS : DWord;
         Responce_VALID : Bool;
         Responce_BUSY : Bool;
         Responce_ERROR : Bool;
         Responce_STATUS : DWord;
         Responce_LEN : Int;
      END_STRUCT;
      Drive_Type_Dummy : Bool;
      Drive_Type_Dummy2 : Bool;
      Response_Format_Dummy : Int;
      Format_Check : Bool;
      Format_Check_1 : Bool;
      Request_Sent_32bit : Bool;
      Request_Sent_16bit : Bool;
      Request_Sent_16bit_1 : Bool;
      RESTART : Bool;
      RESTART_EMG : Bool;
      POWER_RESET_FB_1 : Bool;
   END_VAR
   VAR_TEMP
      PARA_READ_ERR : Int;
      TEMP0 : Time;
      IN_ADDRESS_DW : Word;
      OUT_ADDRESS_DW : Word;
      dummy : Bool;
      MSW_Temp : Struct
         SW : Struct
            AT_SET_POINT : Bool;   // Nopeus asetusarvojen sisällä
            REMONTE : Bool;   // Profibuss ohjaus sallittu
            ABOVE_LIMIT : Bool;   // Nopeus / taajuus yli rajojen
            EXT_CTRL_LOC : Bool;   // 0=EXT1 1=EXT2 selected
            EXT_RUN_ENABLE : Bool;   // Vahinkokäynnistyksen esto
            MSV13 : Bool;   // Ei käytössä
            MSV14 : Bool;   // Ei käytössä
            COOM_FAULT : Bool;   // Kommunikointivika profibus moduuli CH0
            RDY_ON : Bool;   // Käynnistys valmis
            RDY_RUN : Bool;   // Toiminta valmis
            RDY_REF : Bool;   // Käynnissä
            TRIPPED : Bool;   // Häiriö
            OFF2_STATE : Bool;   // Pysäytys vapaasti pyörien
            OFF3_STATE : Bool;   // Pysäytys hahdollisimman nopeasti
            ON_INHIB : Bool;   // Käynnistys estetty
            ALARM : Bool;   // Hälytys
         END_STRUCT;
      END_STRUCT;
      MSW_Conv AT MSW_Temp : Word;
      MCW_Temp : Struct
         CW : Struct
            INCHING_1 : Bool;   // Vakio nopeus ohje 1 käyttöön
            INCHING_2 : Bool;   // Vakio nopeus ohje 2 käyttöön
            REMONTE_CMD : Bool;   // Profibuss ohjaus käyttöön
            EXT_CTRL_LOC : Bool;   // 0=EXT1 1=EXT2 selected
            RESERVE_2 : Bool;   // Ei käytössä
            RESERVE_3 : Bool;   // Ei käytössä
            RESERVE_4 : Bool;   // Ei käytössä
            RESERVE_5 : Bool;   // Ei käytössä
            OFF1 : Bool;   // Käynnistys valmiuteen
            OFF2 : Bool;   // Vapaastipyörien seis
            OFF3 : Bool;   // Hätä-seis pysäytys
            INHIBIT_OPREATION : Bool;   // Käyntiin ohjaus
            RAMP_OUT_ZERO : Bool;   // Ohjauksen vapautus
            RAMP_HOLD : Bool;   // Kiihdytys sallittu
            RAMP_IN_ZERO : Bool;   // Nopeus ohje nollaan
            RESET : Bool;   // Häiriön kuittaus
         END_STRUCT;
      END_STRUCT;
      MCW_Conv AT MCW_Temp : Word;
      "ReadRequest Sent" : Bool;
      PowerState_Temp : Int;
   END_VAR
   VAR_TEMP   // added for the SCL form of the ladder/FBD networks
      _w1 : Bool;
      _w2 : Bool;
      _w3 : Bool;
   END_VAR
BEGIN

REGION Network 1: Set init values
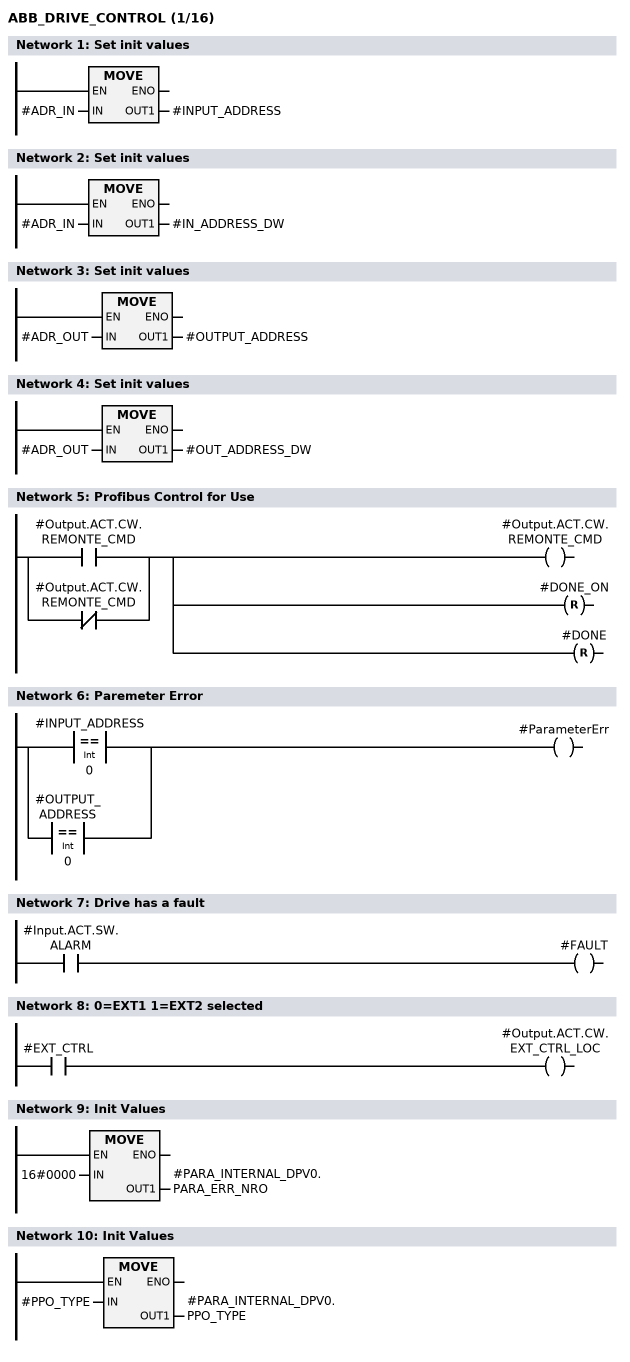
   RUNG wire#powerrail
      { S7_GenerateENO := "TRUE" } Move(in := #ADR_IN, out1 => #INPUT_ADDRESS)
   END_RUNG
   // the same network as SCL:
   #INPUT_ADDRESS := #ADR_IN;
END_REGION

REGION Network 2: Set init values
   RUNG wire#powerrail
      { S7_GenerateENO := "TRUE" } Move(in := #ADR_IN, out1 => #IN_ADDRESS_DW)
   END_RUNG
   // the same network as SCL:
   #IN_ADDRESS_DW := #ADR_IN;
END_REGION

REGION Network 3: Set init values
   RUNG wire#powerrail
      { S7_GenerateENO := "TRUE" } Move(in := #ADR_OUT, out1 => #OUTPUT_ADDRESS)
   END_RUNG
   // the same network as SCL:
   #OUTPUT_ADDRESS := #ADR_OUT;
END_REGION

REGION Network 4: Set init values
   RUNG wire#powerrail
      { S7_GenerateENO := "TRUE" } Move(in := #ADR_OUT, out1 => #OUT_ADDRESS_DW)
   END_RUNG
   // the same network as SCL:
   #OUT_ADDRESS_DW := #ADR_OUT;
END_REGION

REGION Network 5: Profibus Control for Use
   RUNG wire#powerrail
      Contact( #Output.ACT.CW.REMONTE_CMD )
      wire#w1
      Coil( #Output.ACT.CW.REMONTE_CMD )
   END_RUNG
   RUNG wire#powerrail
      I_Contact( #Output.ACT.CW.REMONTE_CMD )
   END_RUNG wire#w1
   RUNG wire#w1
      R_Coil( #DONE_ON )
   END_RUNG
   RUNG wire#w1
      R_Coil( #DONE )
   END_RUNG
   // the same network as SCL:
   #Output.ACT.CW.REMONTE_CMD := #Output.ACT.CW.REMONTE_CMD OR NOT #Output.ACT.CW.REMONTE_CMD;
   IF #Output.ACT.CW.REMONTE_CMD THEN
       #DONE_ON := FALSE;
       #DONE := FALSE;
   END_IF;
END_REGION

REGION Network 6: Paremeter Error
   RUNG wire#powerrail
      { S7_Templates := "SrcType := Int" } EQ_Contact(in1 := #INPUT_ADDRESS, in2 := 0)
      wire#w1
      Coil( #ParameterErr )
   END_RUNG
   RUNG wire#powerrail
      { S7_Templates := "SrcType := Int" } EQ_Contact(in1 := #OUTPUT_ADDRESS, in2 := 0)
   END_RUNG wire#w1
   // the same network as SCL:
   #ParameterErr := (#INPUT_ADDRESS = 0) OR (#OUTPUT_ADDRESS = 0);
END_REGION

REGION Network 7: Drive has a fault
   RUNG wire#powerrail
      Contact( #Input.ACT.SW.ALARM )
      Coil( #FAULT )
   END_RUNG
   // the same network as SCL:
   #FAULT := #Input.ACT.SW.ALARM;
END_REGION

REGION Network 8: 0=EXT1 1=EXT2 selected
   RUNG wire#powerrail
      Contact( #EXT_CTRL )
      Coil( #Output.ACT.CW.EXT_CTRL_LOC )
   END_RUNG
   // the same network as SCL:
   #Output.ACT.CW.EXT_CTRL_LOC := #EXT_CTRL;
END_REGION

REGION Network 9: Init Values
   RUNG wire#powerrail
      { S7_GenerateENO := "TRUE" } Move(in := 16#0000, out1 => #PARA_INTERNAL_DPV0.PARA_ERR_NRO)
   END_RUNG
   // the same network as SCL:
   #PARA_INTERNAL_DPV0.PARA_ERR_NRO := 16#0000;
END_REGION

REGION Network 10: Init Values
   RUNG wire#powerrail
      { S7_GenerateENO := "TRUE" } Move(in := #PPO_TYPE, out1 => #PARA_INTERNAL_DPV0.PPO_TYPE)
   END_RUNG
   // the same network as SCL:
   #PARA_INTERNAL_DPV0.PPO_TYPE := #PPO_TYPE;
END_REGION

REGION Network 11: Init Values
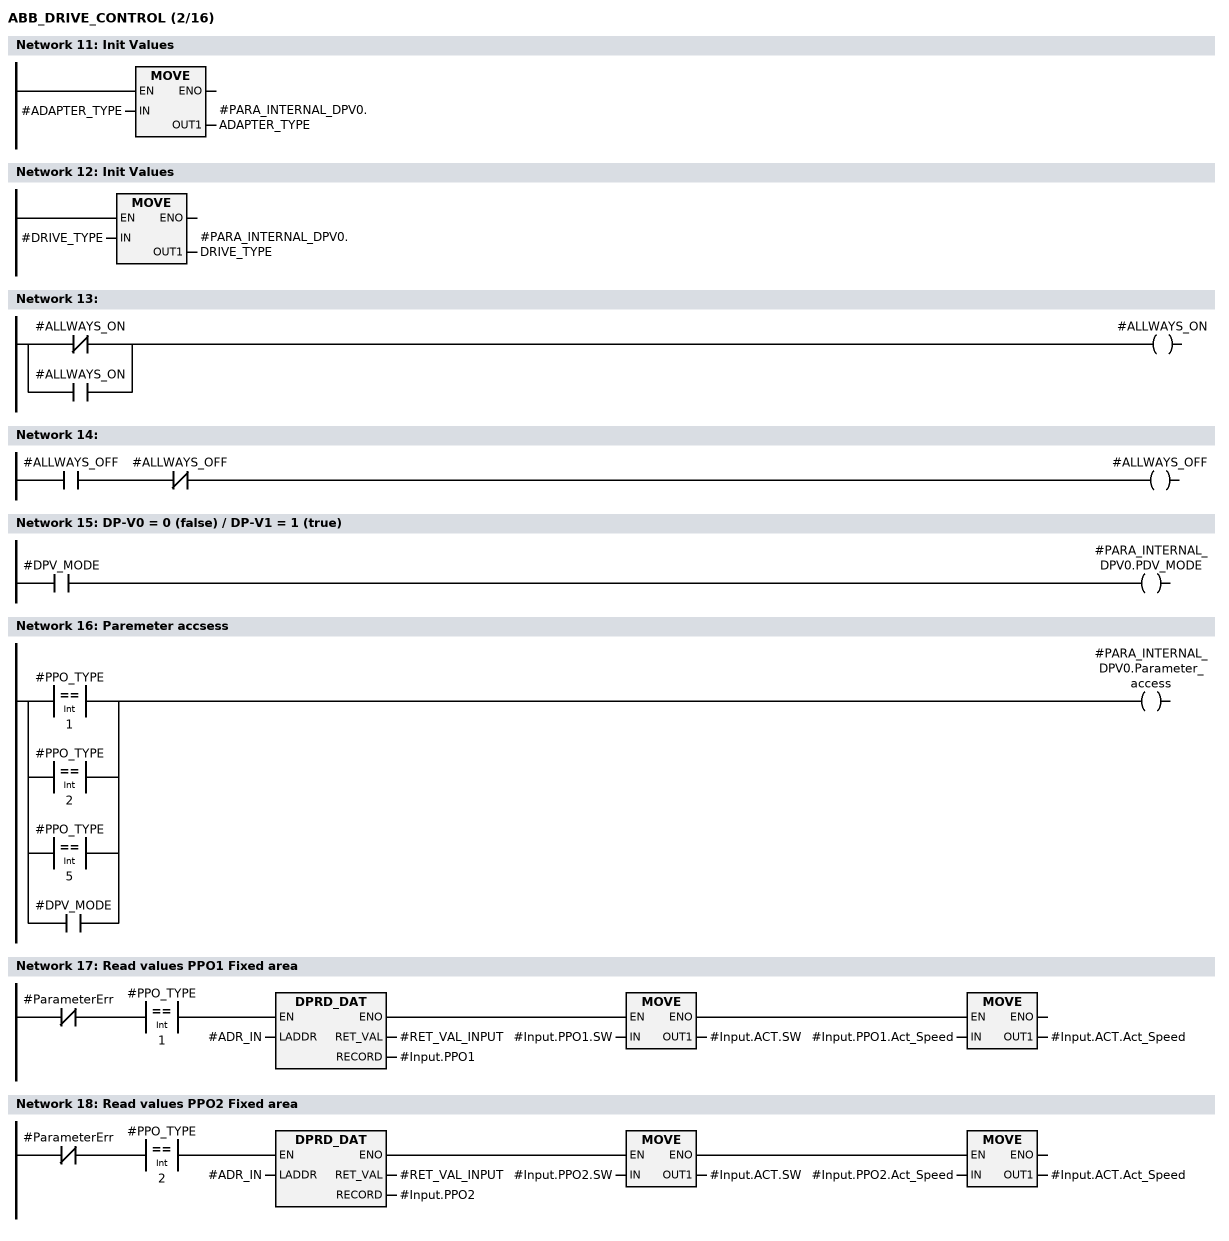
   RUNG wire#powerrail
      { S7_GenerateENO := "TRUE" } Move(in := #ADAPTER_TYPE, out1 => #PARA_INTERNAL_DPV0.ADAPTER_TYPE)
   END_RUNG
   // the same network as SCL:
   #PARA_INTERNAL_DPV0.ADAPTER_TYPE := #ADAPTER_TYPE;
END_REGION

REGION Network 12: Init Values
   RUNG wire#powerrail
      { S7_GenerateENO := "TRUE" } Move(in := #DRIVE_TYPE, out1 => #PARA_INTERNAL_DPV0.DRIVE_TYPE)
   END_RUNG
   // the same network as SCL:
   #PARA_INTERNAL_DPV0.DRIVE_TYPE := #DRIVE_TYPE;
END_REGION

REGION Network 13
   RUNG wire#powerrail
      I_Contact( #ALLWAYS_ON )
      wire#w1
      Coil( #ALLWAYS_ON )
   END_RUNG
   RUNG wire#powerrail
      Contact( #ALLWAYS_ON )
   END_RUNG wire#w1
   // the same network as SCL:
   #ALLWAYS_ON := NOT #ALLWAYS_ON OR #ALLWAYS_ON;
END_REGION

REGION Network 14
   RUNG wire#powerrail
      Contact( #ALLWAYS_OFF )
      I_Contact( #ALLWAYS_OFF )
      Coil( #ALLWAYS_OFF )
   END_RUNG
   // the same network as SCL:
   #ALLWAYS_OFF := #ALLWAYS_OFF AND NOT #ALLWAYS_OFF;
END_REGION

REGION Network 15: DP-V0 = 0 (false) / DP-V1 = 1 (true)
   RUNG wire#powerrail
      Contact( #DPV_MODE )
      Coil( #PARA_INTERNAL_DPV0.PDV_MODE )
   END_RUNG
   // the same network as SCL:
   #PARA_INTERNAL_DPV0.PDV_MODE := #DPV_MODE;
END_REGION

REGION Network 16: Paremeter accsess
   RUNG wire#powerrail
      { S7_Templates := "SrcType := Int" } EQ_Contact(in1 := #PPO_TYPE, in2 := 1)
      wire#w1
      Coil( #PARA_INTERNAL_DPV0.Parameter_access )
   END_RUNG
   RUNG wire#powerrail
      { S7_Templates := "SrcType := Int" } EQ_Contact(in1 := #PPO_TYPE, in2 := 2)
   END_RUNG wire#w1
   RUNG wire#powerrail
      { S7_Templates := "SrcType := Int" } EQ_Contact(in1 := #PPO_TYPE, in2 := 5)
   END_RUNG wire#w1
   RUNG wire#powerrail
      Contact( #DPV_MODE )
   END_RUNG wire#w1
   // the same network as SCL:
   #PARA_INTERNAL_DPV0.Parameter_access := (#PPO_TYPE = 1) OR (#PPO_TYPE = 2) OR (#PPO_TYPE = 5) OR #DPV_MODE;
END_REGION

REGION Network 17: Read values PPO1 Fixed area
   // ENO of a box is taken as its EN; it also drops when the box reports an error
   IF NOT #ParameterErr AND (#PPO_TYPE = 1) THEN
       #RET_VAL_INPUT := DPRD_DAT(LADDR := #ADR_IN, RECORD => #Input.PPO1);
       #Input.ACT.SW := #Input.PPO1.SW;
       #Input.ACT.Act_Speed := #Input.PPO1.Act_Speed;
   END_IF;
END_REGION

REGION Network 18: Read values PPO2 Fixed area
   // ENO of a box is taken as its EN; it also drops when the box reports an error
   IF NOT #ParameterErr AND (#PPO_TYPE = 2) THEN
       #RET_VAL_INPUT := DPRD_DAT(LADDR := #ADR_IN, RECORD => #Input.PPO2);
       #Input.ACT.SW := #Input.PPO2.SW;
       #Input.ACT.Act_Speed := #Input.PPO2.Act_Speed;
   END_IF;
END_REGION

REGION Network 19: Move PPO2 Process data area
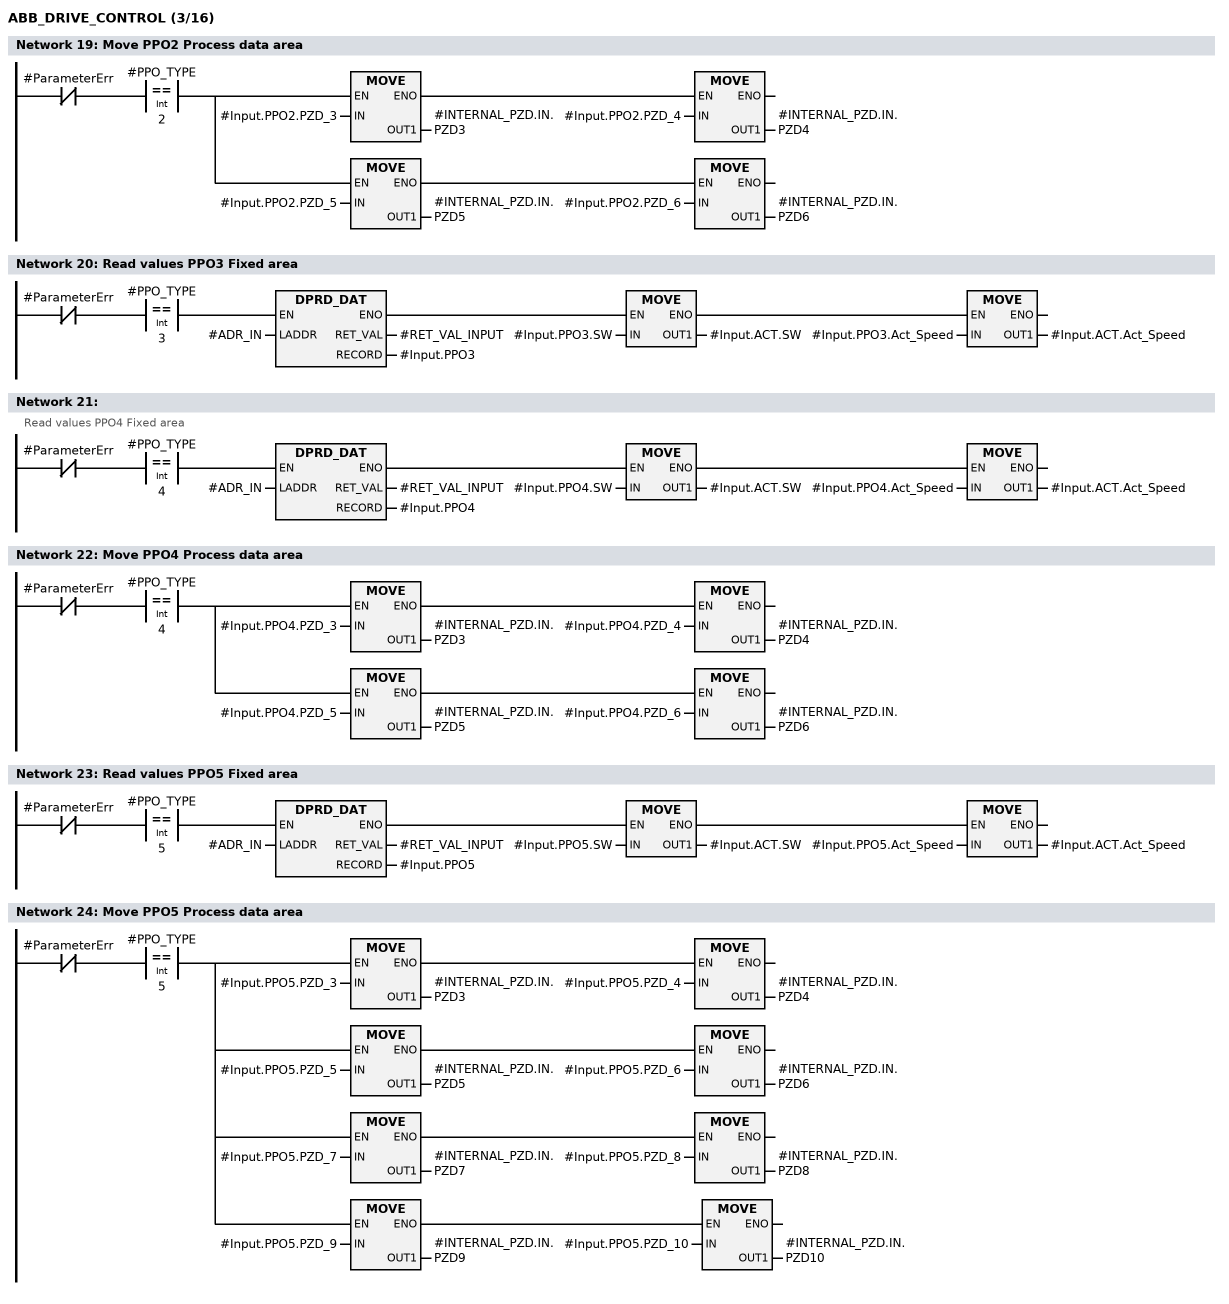
   RUNG wire#powerrail
      I_Contact( #ParameterErr )
      { S7_Templates := "SrcType := Int" } EQ_Contact(in1 := #PPO_TYPE, in2 := 2)
      wire#w1
      { S7_GenerateENO := "TRUE" } Move(in := #Input.PPO2.PZD_3, out1 => #INTERNAL_PZD.IN.PZD3)
      { S7_GenerateENO := "TRUE" } Move(in := #Input.PPO2.PZD_4, out1 => #INTERNAL_PZD.IN.PZD4)
   END_RUNG
   RUNG wire#w1
      { S7_GenerateENO := "TRUE" } Move(in := #Input.PPO2.PZD_5, out1 => #INTERNAL_PZD.IN.PZD5)
      { S7_GenerateENO := "TRUE" } Move(in := #Input.PPO2.PZD_6, out1 => #INTERNAL_PZD.IN.PZD6)
   END_RUNG
   // the same network as SCL:
   // ENO of a box is taken as its EN; it also drops when the box reports an error
   IF NOT #ParameterErr AND (#PPO_TYPE = 2) THEN
       #INTERNAL_PZD.IN.PZD3 := #Input.PPO2.PZD_3;
       #INTERNAL_PZD.IN.PZD4 := #Input.PPO2.PZD_4;
       #INTERNAL_PZD.IN.PZD5 := #Input.PPO2.PZD_5;
       #INTERNAL_PZD.IN.PZD6 := #Input.PPO2.PZD_6;
   END_IF;
END_REGION

REGION Network 20: Read values PPO3 Fixed area
   // ENO of a box is taken as its EN; it also drops when the box reports an error
   IF NOT #ParameterErr AND (#PPO_TYPE = 3) THEN
       #RET_VAL_INPUT := DPRD_DAT(LADDR := #ADR_IN, RECORD => #Input.PPO3);
       #Input.ACT.SW := #Input.PPO3.SW;
       #Input.ACT.Act_Speed := #Input.PPO3.Act_Speed;
   END_IF;
END_REGION

REGION Network 21
   // Read values PPO4 Fixed area
   // ENO of a box is taken as its EN; it also drops when the box reports an error
   IF NOT #ParameterErr AND (#PPO_TYPE = 4) THEN
       #RET_VAL_INPUT := DPRD_DAT(LADDR := #ADR_IN, RECORD => #Input.PPO4);
       #Input.ACT.SW := #Input.PPO4.SW;
       #Input.ACT.Act_Speed := #Input.PPO4.Act_Speed;
   END_IF;
END_REGION

REGION Network 22: Move PPO4 Process data area
   RUNG wire#powerrail
      I_Contact( #ParameterErr )
      { S7_Templates := "SrcType := Int" } EQ_Contact(in1 := #PPO_TYPE, in2 := 4)
      wire#w1
      { S7_GenerateENO := "TRUE" } Move(in := #Input.PPO4.PZD_3, out1 => #INTERNAL_PZD.IN.PZD3)
      { S7_GenerateENO := "TRUE" } Move(in := #Input.PPO4.PZD_4, out1 => #INTERNAL_PZD.IN.PZD4)
   END_RUNG
   RUNG wire#w1
      { S7_GenerateENO := "TRUE" } Move(in := #Input.PPO4.PZD_5, out1 => #INTERNAL_PZD.IN.PZD5)
      { S7_GenerateENO := "TRUE" } Move(in := #Input.PPO4.PZD_6, out1 => #INTERNAL_PZD.IN.PZD6)
   END_RUNG
   // the same network as SCL:
   // ENO of a box is taken as its EN; it also drops when the box reports an error
   IF NOT #ParameterErr AND (#PPO_TYPE = 4) THEN
       #INTERNAL_PZD.IN.PZD3 := #Input.PPO4.PZD_3;
       #INTERNAL_PZD.IN.PZD4 := #Input.PPO4.PZD_4;
       #INTERNAL_PZD.IN.PZD5 := #Input.PPO4.PZD_5;
       #INTERNAL_PZD.IN.PZD6 := #Input.PPO4.PZD_6;
   END_IF;
END_REGION

REGION Network 23: Read values PPO5 Fixed area
   // ENO of a box is taken as its EN; it also drops when the box reports an error
   IF NOT #ParameterErr AND (#PPO_TYPE = 5) THEN
       #RET_VAL_INPUT := DPRD_DAT(LADDR := #ADR_IN, RECORD => #Input.PPO5);
       #Input.ACT.SW := #Input.PPO5.SW;
       #Input.ACT.Act_Speed := #Input.PPO5.Act_Speed;
   END_IF;
END_REGION

REGION Network 24: Move PPO5 Process data area
   RUNG wire#powerrail
      I_Contact( #ParameterErr )
      { S7_Templates := "SrcType := Int" } EQ_Contact(in1 := #PPO_TYPE, in2 := 5)
      wire#w1
      { S7_GenerateENO := "TRUE" } Move(in := #Input.PPO5.PZD_3, out1 => #INTERNAL_PZD.IN.PZD3)
      { S7_GenerateENO := "TRUE" } Move(in := #Input.PPO5.PZD_4, out1 => #INTERNAL_PZD.IN.PZD4)
   END_RUNG
   RUNG wire#w1
      { S7_GenerateENO := "TRUE" } Move(in := #Input.PPO5.PZD_5, out1 => #INTERNAL_PZD.IN.PZD5)
      { S7_GenerateENO := "TRUE" } Move(in := #Input.PPO5.PZD_6, out1 => #INTERNAL_PZD.IN.PZD6)
   END_RUNG
   RUNG wire#w1
      { S7_GenerateENO := "TRUE" } Move(in := #Input.PPO5.PZD_7, out1 => #INTERNAL_PZD.IN.PZD7)
      { S7_GenerateENO := "TRUE" } Move(in := #Input.PPO5.PZD_8, out1 => #INTERNAL_PZD.IN.PZD8)
   END_RUNG
   RUNG wire#w1
      { S7_GenerateENO := "TRUE" } Move(in := #Input.PPO5.PZD_9, out1 => #INTERNAL_PZD.IN.PZD9)
      { S7_GenerateENO := "TRUE" } Move(in := #Input.PPO5.PZD_10, out1 => #INTERNAL_PZD.IN.PZD10)
   END_RUNG
   // the same network as SCL:
   // ENO of a box is taken as its EN; it also drops when the box reports an error
   IF NOT #ParameterErr AND (#PPO_TYPE = 5) THEN
       #INTERNAL_PZD.IN.PZD3 := #Input.PPO5.PZD_3;
       #INTERNAL_PZD.IN.PZD4 := #Input.PPO5.PZD_4;
       #INTERNAL_PZD.IN.PZD5 := #Input.PPO5.PZD_5;
       #INTERNAL_PZD.IN.PZD6 := #Input.PPO5.PZD_6;
       #INTERNAL_PZD.IN.PZD7 := #Input.PPO5.PZD_7;
       #INTERNAL_PZD.IN.PZD8 := #Input.PPO5.PZD_8;
       #INTERNAL_PZD.IN.PZD9 := #Input.PPO5.PZD_9;
       #INTERNAL_PZD.IN.PZD10 := #Input.PPO5.PZD_10;
   END_IF;
END_REGION

REGION Network 25: Read values PPO6 Fixed area
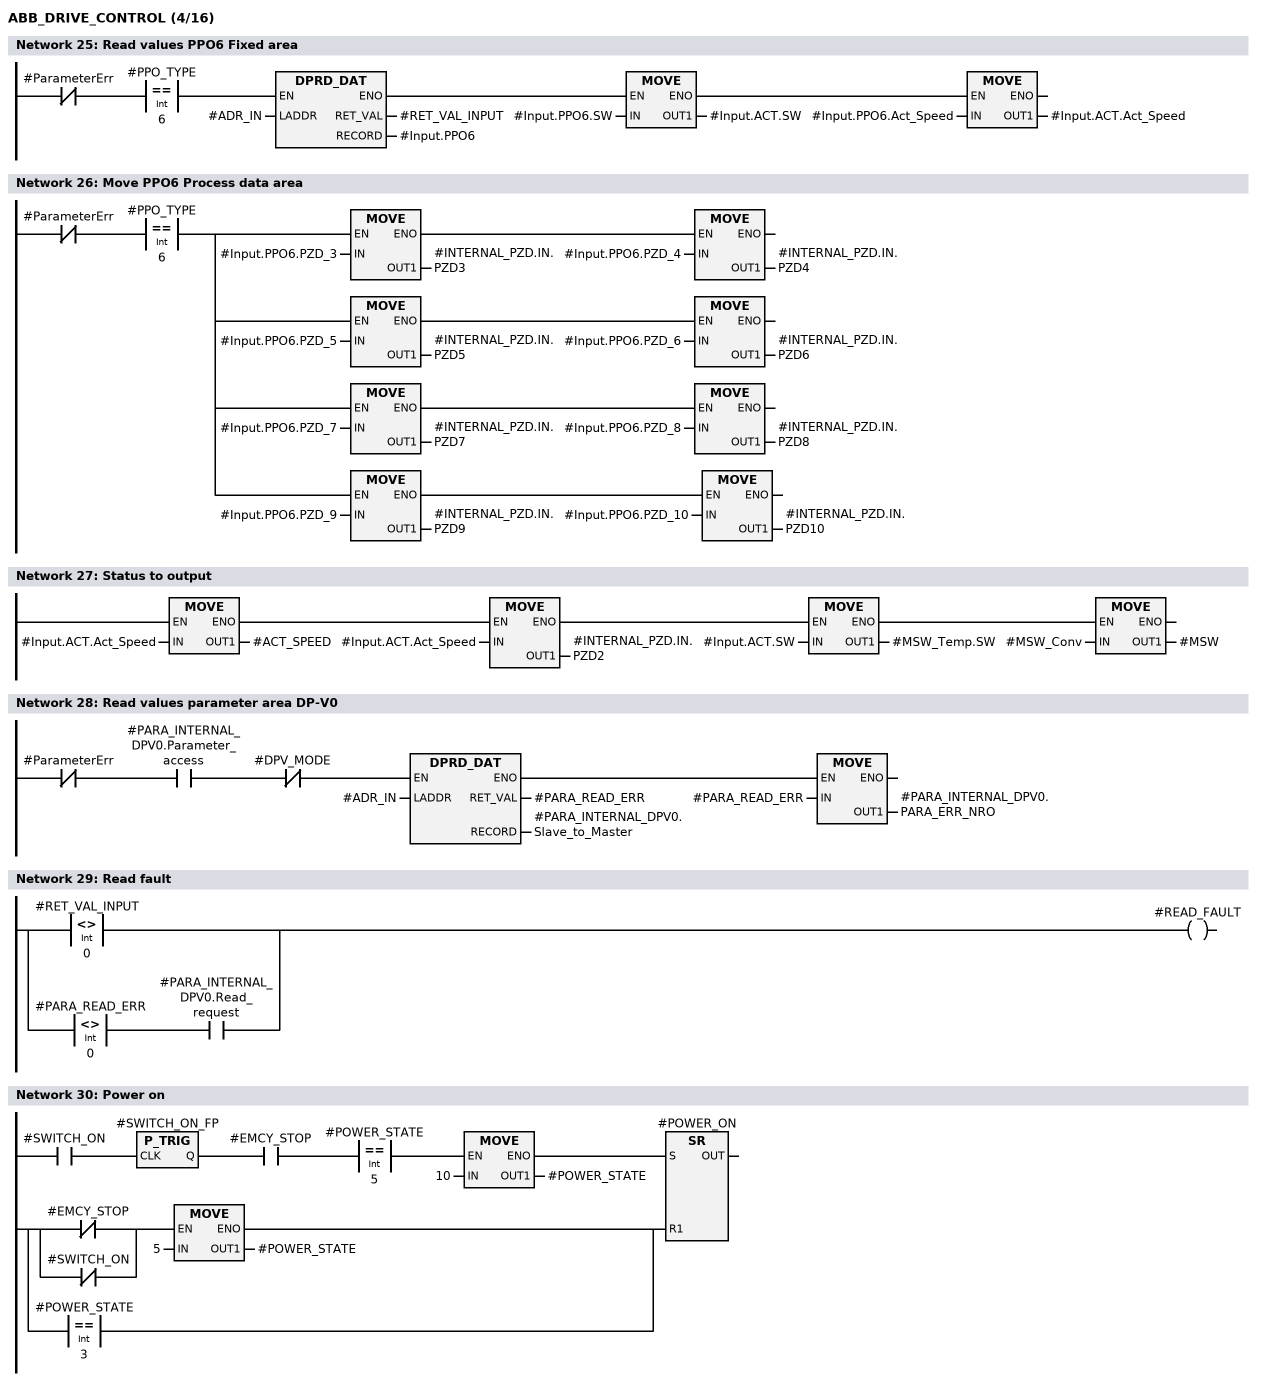
   // ENO of a box is taken as its EN; it also drops when the box reports an error
   IF NOT #ParameterErr AND (#PPO_TYPE = 6) THEN
       #RET_VAL_INPUT := DPRD_DAT(LADDR := #ADR_IN, RECORD => #Input.PPO6);
       #Input.ACT.SW := #Input.PPO6.SW;
       #Input.ACT.Act_Speed := #Input.PPO6.Act_Speed;
   END_IF;
END_REGION

REGION Network 26: Move PPO6 Process data area
   RUNG wire#powerrail
      I_Contact( #ParameterErr )
      { S7_Templates := "SrcType := Int" } EQ_Contact(in1 := #PPO_TYPE, in2 := 6)
      wire#w1
      { S7_GenerateENO := "TRUE" } Move(in := #Input.PPO6.PZD_3, out1 => #INTERNAL_PZD.IN.PZD3)
      { S7_GenerateENO := "TRUE" } Move(in := #Input.PPO6.PZD_4, out1 => #INTERNAL_PZD.IN.PZD4)
   END_RUNG
   RUNG wire#w1
      { S7_GenerateENO := "TRUE" } Move(in := #Input.PPO6.PZD_5, out1 => #INTERNAL_PZD.IN.PZD5)
      { S7_GenerateENO := "TRUE" } Move(in := #Input.PPO6.PZD_6, out1 => #INTERNAL_PZD.IN.PZD6)
   END_RUNG
   RUNG wire#w1
      { S7_GenerateENO := "TRUE" } Move(in := #Input.PPO6.PZD_7, out1 => #INTERNAL_PZD.IN.PZD7)
      { S7_GenerateENO := "TRUE" } Move(in := #Input.PPO6.PZD_8, out1 => #INTERNAL_PZD.IN.PZD8)
   END_RUNG
   RUNG wire#w1
      { S7_GenerateENO := "TRUE" } Move(in := #Input.PPO6.PZD_9, out1 => #INTERNAL_PZD.IN.PZD9)
      { S7_GenerateENO := "TRUE" } Move(in := #Input.PPO6.PZD_10, out1 => #INTERNAL_PZD.IN.PZD10)
   END_RUNG
   // the same network as SCL:
   // ENO of a box is taken as its EN; it also drops when the box reports an error
   IF NOT #ParameterErr AND (#PPO_TYPE = 6) THEN
       #INTERNAL_PZD.IN.PZD3 := #Input.PPO6.PZD_3;
       #INTERNAL_PZD.IN.PZD4 := #Input.PPO6.PZD_4;
       #INTERNAL_PZD.IN.PZD5 := #Input.PPO6.PZD_5;
       #INTERNAL_PZD.IN.PZD6 := #Input.PPO6.PZD_6;
       #INTERNAL_PZD.IN.PZD7 := #Input.PPO6.PZD_7;
       #INTERNAL_PZD.IN.PZD8 := #Input.PPO6.PZD_8;
       #INTERNAL_PZD.IN.PZD9 := #Input.PPO6.PZD_9;
       #INTERNAL_PZD.IN.PZD10 := #Input.PPO6.PZD_10;
   END_IF;
END_REGION

REGION Network 27: Status to output
   RUNG wire#powerrail
      { S7_GenerateENO := "TRUE" } Move(in := #Input.ACT.Act_Speed, out1 => #ACT_SPEED)
      { S7_GenerateENO := "TRUE" } Move(in := #Input.ACT.Act_Speed, out1 => #INTERNAL_PZD.IN.PZD2)
      { S7_GenerateENO := "TRUE" } Move(in := #Input.ACT.SW, out1 => #MSW_Temp.SW)
      { S7_GenerateENO := "TRUE" } Move(in := #MSW_Conv, out1 => #MSW)
   END_RUNG
   // the same network as SCL:
   // ENO of a box is taken as its EN; it also drops when the box reports an error
   #ACT_SPEED := #Input.ACT.Act_Speed;
   #INTERNAL_PZD.IN.PZD2 := #Input.ACT.Act_Speed;
   #MSW_Temp.SW := #Input.ACT.SW;
   #MSW := #MSW_Conv;
END_REGION

REGION Network 28: Read values parameter area DP-V0
   // ENO of a box is taken as its EN; it also drops when the box reports an error
   IF NOT #ParameterErr AND #PARA_INTERNAL_DPV0.Parameter_access AND NOT #DPV_MODE THEN
       #PARA_READ_ERR := DPRD_DAT(LADDR := #ADR_IN, RECORD => #PARA_INTERNAL_DPV0.Slave_to_Master);
       #PARA_INTERNAL_DPV0.PARA_ERR_NRO := #PARA_READ_ERR;
   END_IF;
END_REGION

REGION Network 29: Read fault
   RUNG wire#powerrail
      { S7_Templates := "SrcType := Int" } NE_Contact(in1 := #RET_VAL_INPUT, in2 := 0)
      wire#w1
      Coil( #READ_FAULT )
   END_RUNG
   RUNG wire#powerrail
      { S7_Templates := "SrcType := Int" } NE_Contact(in1 := #PARA_READ_ERR, in2 := 0)
      Contact( #PARA_INTERNAL_DPV0.Read_request )
   END_RUNG wire#w1
   // the same network as SCL:
   #READ_FAULT := (#RET_VAL_INPUT <> 0) OR ((#PARA_READ_ERR <> 0) AND #PARA_INTERNAL_DPV0.Read_request);
END_REGION

REGION Network 30: Power on
   RUNG wire#powerrail
      Contact( #SWITCH_ON )
      P_Trig( #SWITCH_ON_FP )
      Contact( #EMCY_STOP )
      { S7_Templates := "SrcType := Int" } EQ_Contact(in1 := #POWER_STATE, in2 := 5)
      { S7_GenerateENO := "TRUE" } Move(in := 10, out1 => #POWER_STATE)
      S_SR(operand := #POWER_ON, r1 := wire#w2)
   END_RUNG
   RUNG wire#powerrail
      I_Contact( #EMCY_STOP )
      wire#w1
      { S7_GenerateENO := "TRUE" } Move(in := 5, out1 => #POWER_STATE)
   END_RUNG wire#w2
   RUNG wire#powerrail
      I_Contact( #SWITCH_ON )
   END_RUNG wire#w1
   RUNG wire#powerrail
      { S7_Templates := "SrcType := Int" } EQ_Contact(in1 := #POWER_STATE, in2 := 3)
   END_RUNG wire#w2
   // the same network as SCL:
   // ENO of a box is taken as its EN; it also drops when the box reports an error
   #_w1 := #SWITCH_ON AND NOT #SWITCH_ON_FP;   // rising edge
   #SWITCH_ON_FP := #SWITCH_ON;
   #_w2 := #_w1 AND #EMCY_STOP AND (#POWER_STATE = 5);
   IF #_w2 THEN #POWER_STATE := 10; END_IF;
   #_w3 := NOT #EMCY_STOP OR NOT #SWITCH_ON;
   IF #_w3 THEN #POWER_STATE := 5; END_IF;
   IF #_w2 THEN
       #POWER_ON := TRUE;   // SR flip-flop
   END_IF;
   IF #_w3 OR (#POWER_STATE = 3) THEN #POWER_ON := FALSE; END_IF;
END_REGION

REGION Network 31: Power state
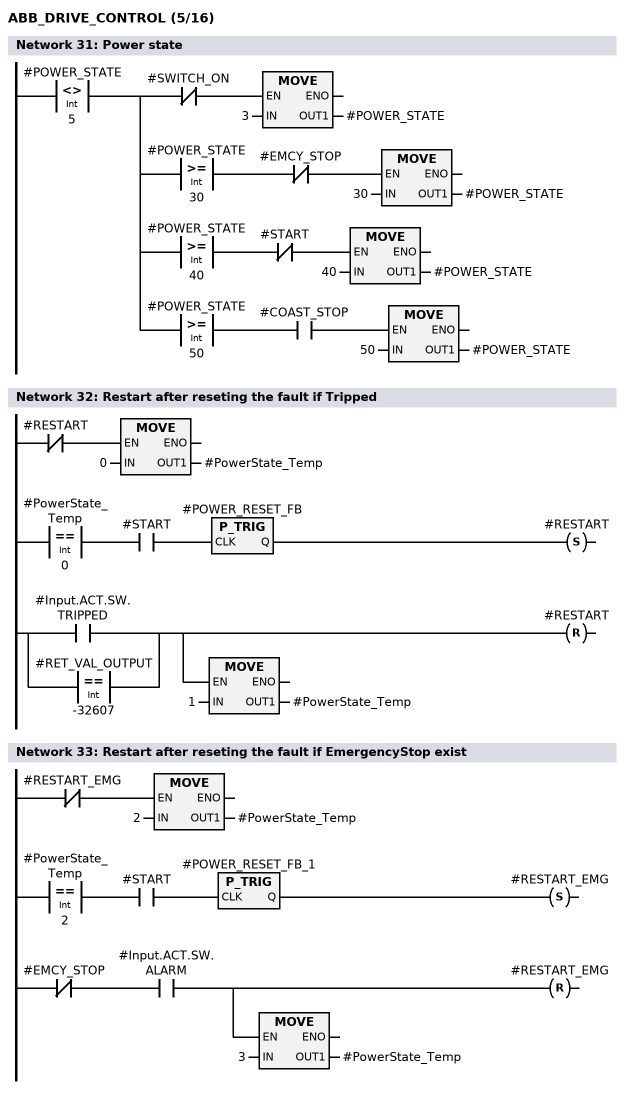
   RUNG wire#powerrail
      { S7_Templates := "SrcType := Int" } NE_Contact(in1 := #POWER_STATE, in2 := 5)
      wire#w1
      I_Contact( #SWITCH_ON )
      { S7_GenerateENO := "TRUE" } Move(in := 3, out1 => #POWER_STATE)
   END_RUNG
   RUNG wire#w1
      { S7_Templates := "SrcType := Int" } GE_Contact(in1 := #POWER_STATE, in2 := 30)
      I_Contact( #EMCY_STOP )
      { S7_GenerateENO := "TRUE" } Move(in := 30, out1 => #POWER_STATE)
   END_RUNG
   RUNG wire#w1
      { S7_Templates := "SrcType := Int" } GE_Contact(in1 := #POWER_STATE, in2 := 40)
      I_Contact( #START )
      { S7_GenerateENO := "TRUE" } Move(in := 40, out1 => #POWER_STATE)
   END_RUNG
   RUNG wire#w1
      { S7_Templates := "SrcType := Int" } GE_Contact(in1 := #POWER_STATE, in2 := 50)
      Contact( #COAST_STOP )
      { S7_GenerateENO := "TRUE" } Move(in := 50, out1 => #POWER_STATE)
   END_RUNG
   // the same network as SCL:
   #_w1 := #POWER_STATE <> 5;
   IF #_w1 AND NOT #SWITCH_ON THEN #POWER_STATE := 3; END_IF;
   IF #_w1 AND (#POWER_STATE >= 30) AND NOT #EMCY_STOP THEN #POWER_STATE := 30; END_IF;
   IF #_w1 AND (#POWER_STATE >= 40) AND NOT #START THEN #POWER_STATE := 40; END_IF;
   IF #_w1 AND (#POWER_STATE >= 50) AND #COAST_STOP THEN #POWER_STATE := 50; END_IF;
END_REGION

REGION Network 32: Restart after reseting the fault if Tripped
   RUNG wire#powerrail
      I_Contact( #RESTART )
      Move(in := 0, out1 => #PowerState_Temp)
   END_RUNG
   RUNG wire#powerrail
      { S7_Templates := "SrcType := Int" } EQ_Contact(in1 := #PowerState_Temp, in2 := 0)
      Contact( #START )
      P_Trig( #POWER_RESET_FB )
      S_Coil( #RESTART )
   END_RUNG
   RUNG wire#powerrail
      Contact( #Input.ACT.SW.TRIPPED )
      wire#w1
      R_Coil( #RESTART )
   END_RUNG
   RUNG wire#powerrail
      { S7_Templates := "SrcType := Int" } EQ_Contact(in1 := #RET_VAL_OUTPUT, in2 := -32607)
   END_RUNG wire#w1
   RUNG wire#w1
      Move(in := 1, out1 => #PowerState_Temp)
   END_RUNG
   // the same network as SCL:
   IF NOT #RESTART THEN #PowerState_Temp := 0; END_IF;
   #_w1 := (#PowerState_Temp = 0) AND #START;
   #_w2 := #_w1 AND NOT #POWER_RESET_FB;   // rising edge
   #POWER_RESET_FB := #_w1;
   IF #_w2 THEN #RESTART := TRUE; END_IF;
   IF #Input.ACT.SW.TRIPPED OR (#RET_VAL_OUTPUT = (-32607)) THEN
       #RESTART := FALSE;
       #PowerState_Temp := 1;
   END_IF;
END_REGION

REGION Network 33: Restart after reseting the fault if EmergencyStop exist
   RUNG wire#powerrail
      I_Contact( #RESTART_EMG )
      Move(in := 2, out1 => #PowerState_Temp)
   END_RUNG
   RUNG wire#powerrail
      { S7_Templates := "SrcType := Int" } EQ_Contact(in1 := #PowerState_Temp, in2 := 2)
      Contact( #START )
      P_Trig( #POWER_RESET_FB_1 )
      S_Coil( #RESTART_EMG )
   END_RUNG
   RUNG wire#powerrail
      I_Contact( #EMCY_STOP )
      Contact( #Input.ACT.SW.ALARM )
      wire#w1
      R_Coil( #RESTART_EMG )
   END_RUNG
   RUNG wire#w1
      Move(in := 3, out1 => #PowerState_Temp)
   END_RUNG
   // the same network as SCL:
   IF NOT #RESTART_EMG THEN #PowerState_Temp := 2; END_IF;
   #_w1 := (#PowerState_Temp = 2) AND #START;
   #_w2 := #_w1 AND NOT #POWER_RESET_FB_1;   // rising edge
   #POWER_RESET_FB_1 := #_w1;
   IF #_w2 THEN #RESTART_EMG := TRUE; END_IF;
   IF NOT #EMCY_STOP AND #Input.ACT.SW.ALARM THEN
       #RESTART_EMG := FALSE;
       #PowerState_Temp := 3;
   END_IF;
END_REGION

REGION Network 34: Switch off state -> wait for start
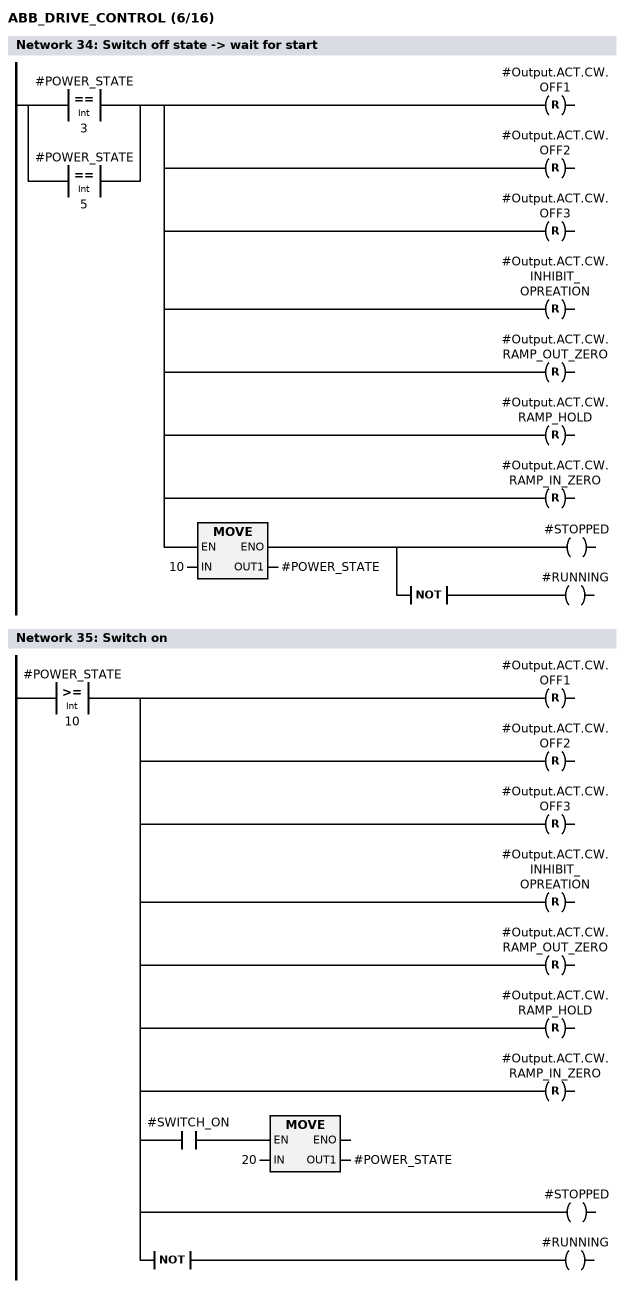
   RUNG wire#powerrail
      { S7_Templates := "SrcType := Int" } EQ_Contact(in1 := #POWER_STATE, in2 := 3)
      wire#w1
      R_Coil( #Output.ACT.CW.OFF1 )
   END_RUNG
   RUNG wire#powerrail
      { S7_Templates := "SrcType := Int" } EQ_Contact(in1 := #POWER_STATE, in2 := 5)
   END_RUNG wire#w1
   RUNG wire#w1
      R_Coil( #Output.ACT.CW.OFF2 )
   END_RUNG
   RUNG wire#w1
      R_Coil( #Output.ACT.CW.OFF3 )
   END_RUNG
   RUNG wire#w1
      R_Coil( #Output.ACT.CW.INHIBIT_OPREATION )
   END_RUNG
   RUNG wire#w1
      R_Coil( #Output.ACT.CW.RAMP_OUT_ZERO )
   END_RUNG
   RUNG wire#w1
      R_Coil( #Output.ACT.CW.RAMP_HOLD )
   END_RUNG
   RUNG wire#w1
      R_Coil( #Output.ACT.CW.RAMP_IN_ZERO )
   END_RUNG
   RUNG wire#w1
      { S7_GenerateENO := "TRUE" } Move(in := 10, out1 => #POWER_STATE)
      wire#w2
      Coil( #STOPPED )
   END_RUNG
   RUNG wire#w2
      Not()
      Coil( #RUNNING )
   END_RUNG
   // the same network as SCL:
   // ENO of a box is taken as its EN; it also drops when the box reports an error
   #_w1 := (#POWER_STATE = 3) OR (#POWER_STATE = 5);
   IF #_w1 THEN
       #Output.ACT.CW.OFF1 := FALSE;
       #Output.ACT.CW.OFF2 := FALSE;
       #Output.ACT.CW.OFF3 := FALSE;
       #Output.ACT.CW.INHIBIT_OPREATION := FALSE;
       #Output.ACT.CW.RAMP_OUT_ZERO := FALSE;
       #Output.ACT.CW.RAMP_HOLD := FALSE;
       #Output.ACT.CW.RAMP_IN_ZERO := FALSE;
       #POWER_STATE := 10;
   END_IF;
   #STOPPED := #_w1;
   #RUNNING := NOT #_w1;
END_REGION

REGION Network 35: Switch on
   RUNG wire#powerrail
      { S7_Templates := "SrcType := Int" } GE_Contact(in1 := #POWER_STATE, in2 := 10)
      wire#w1
      R_Coil( #Output.ACT.CW.OFF1 )
   END_RUNG
   RUNG wire#w1
      R_Coil( #Output.ACT.CW.OFF2 )
   END_RUNG
   RUNG wire#w1
      R_Coil( #Output.ACT.CW.OFF3 )
   END_RUNG
   RUNG wire#w1
      R_Coil( #Output.ACT.CW.INHIBIT_OPREATION )
   END_RUNG
   RUNG wire#w1
      R_Coil( #Output.ACT.CW.RAMP_OUT_ZERO )
   END_RUNG
   RUNG wire#w1
      R_Coil( #Output.ACT.CW.RAMP_HOLD )
   END_RUNG
   RUNG wire#w1
      R_Coil( #Output.ACT.CW.RAMP_IN_ZERO )
   END_RUNG
   RUNG wire#w1
      Contact( #SWITCH_ON )
      { S7_GenerateENO := "TRUE" } Move(in := 20, out1 => #POWER_STATE)
   END_RUNG
   RUNG wire#w1
      Coil( #STOPPED )
   END_RUNG
   RUNG wire#w1
      Not()
      Coil( #RUNNING )
   END_RUNG
   // the same network as SCL:
   #_w1 := #POWER_STATE >= 10;
   IF #_w1 THEN
       #Output.ACT.CW.OFF1 := FALSE;
       #Output.ACT.CW.OFF2 := FALSE;
       #Output.ACT.CW.OFF3 := FALSE;
       #Output.ACT.CW.INHIBIT_OPREATION := FALSE;
       #Output.ACT.CW.RAMP_OUT_ZERO := FALSE;
       #Output.ACT.CW.RAMP_HOLD := FALSE;
       #Output.ACT.CW.RAMP_IN_ZERO := FALSE;
   END_IF;
   IF #_w1 AND #SWITCH_ON THEN #POWER_STATE := 20; END_IF;
   #STOPPED := #_w1;
   #RUNNING := NOT #_w1;
END_REGION

REGION Network 36: Future use
END_REGION

REGION Network 37: OFF2
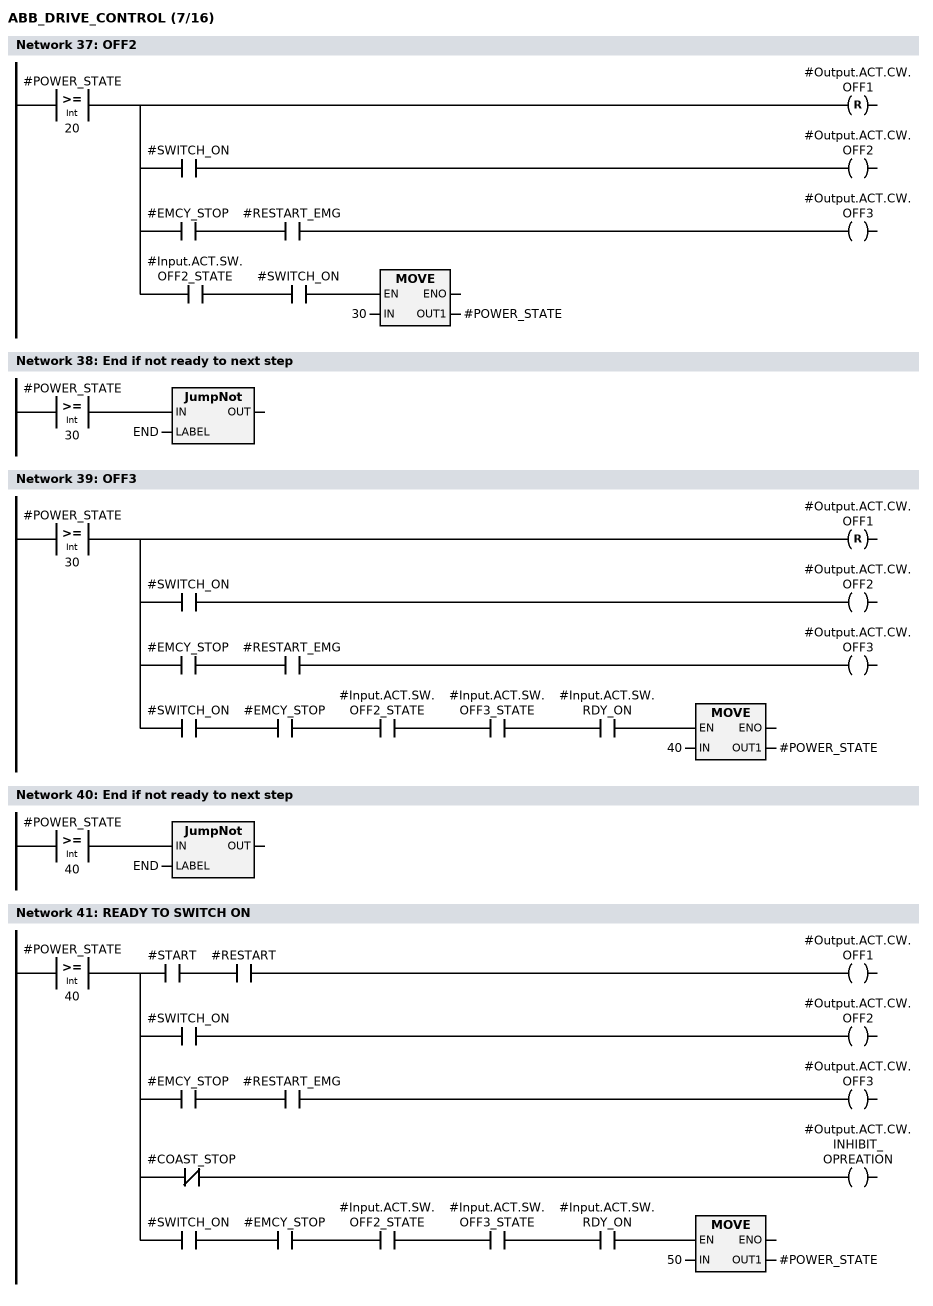
   RUNG wire#powerrail
      { S7_Templates := "SrcType := Int" } GE_Contact(in1 := #POWER_STATE, in2 := 20)
      wire#w1
      R_Coil( #Output.ACT.CW.OFF1 )
   END_RUNG
   RUNG wire#w1
      Contact( #SWITCH_ON )
      Coil( #Output.ACT.CW.OFF2 )
   END_RUNG
   RUNG wire#w1
      Contact( #EMCY_STOP )
      Contact( #RESTART_EMG )
      Coil( #Output.ACT.CW.OFF3 )
   END_RUNG
   RUNG wire#w1
      Contact( #Input.ACT.SW.OFF2_STATE )
      Contact( #SWITCH_ON )
      { S7_GenerateENO := "TRUE" } Move(in := 30, out1 => #POWER_STATE)
   END_RUNG
   // the same network as SCL:
   #_w1 := #POWER_STATE >= 20;
   IF #_w1 THEN #Output.ACT.CW.OFF1 := FALSE; END_IF;
   #Output.ACT.CW.OFF2 := #_w1 AND #SWITCH_ON;
   #Output.ACT.CW.OFF3 := #_w1 AND #EMCY_STOP AND #RESTART_EMG;
   IF #_w1 AND #Input.ACT.SW.OFF2_STATE AND #SWITCH_ON THEN #POWER_STATE := 30; END_IF;
END_REGION

REGION Network 38: End if not ready to next step
   // no SCL statement known for JumpNot: written as a call
   JumpNot(in := #POWER_STATE >= 30, label := END);
END_REGION

REGION Network 39: OFF3
   RUNG wire#powerrail
      { S7_Templates := "SrcType := Int" } GE_Contact(in1 := #POWER_STATE, in2 := 30)
      wire#w1
      R_Coil( #Output.ACT.CW.OFF1 )
   END_RUNG
   RUNG wire#w1
      Contact( #SWITCH_ON )
      Coil( #Output.ACT.CW.OFF2 )
   END_RUNG
   RUNG wire#w1
      Contact( #EMCY_STOP )
      Contact( #RESTART_EMG )
      Coil( #Output.ACT.CW.OFF3 )
   END_RUNG
   RUNG wire#w1
      Contact( #SWITCH_ON )
      Contact( #EMCY_STOP )
      Contact( #Input.ACT.SW.OFF2_STATE )
      Contact( #Input.ACT.SW.OFF3_STATE )
      Contact( #Input.ACT.SW.RDY_ON )
      { S7_GenerateENO := "TRUE" } Move(in := 40, out1 => #POWER_STATE)
   END_RUNG
   // the same network as SCL:
   #_w1 := #POWER_STATE >= 30;
   IF #_w1 THEN #Output.ACT.CW.OFF1 := FALSE; END_IF;
   #Output.ACT.CW.OFF2 := #_w1 AND #SWITCH_ON;
   #Output.ACT.CW.OFF3 := #_w1 AND #EMCY_STOP AND #RESTART_EMG;
   IF #_w1 AND #SWITCH_ON AND #EMCY_STOP AND #Input.ACT.SW.OFF2_STATE AND #Input.ACT.SW.OFF3_STATE AND #Input.ACT.SW.RDY_ON THEN
       #POWER_STATE := 40;
   END_IF;
END_REGION

REGION Network 40: End if not ready to next step
   // no SCL statement known for JumpNot: written as a call
   JumpNot(in := #POWER_STATE >= 40, label := END);
END_REGION

REGION Network 41: READY TO SWITCH ON
   RUNG wire#powerrail
      { S7_Templates := "SrcType := Int" } GE_Contact(in1 := #POWER_STATE, in2 := 40)
      wire#w1
      Contact( #START )
      Contact( #RESTART )
      Coil( #Output.ACT.CW.OFF1 )
   END_RUNG
   RUNG wire#w1
      Contact( #SWITCH_ON )
      Coil( #Output.ACT.CW.OFF2 )
   END_RUNG
   RUNG wire#w1
      Contact( #EMCY_STOP )
      Contact( #RESTART_EMG )
      Coil( #Output.ACT.CW.OFF3 )
   END_RUNG
   RUNG wire#w1
      I_Contact( #COAST_STOP )
      Coil( #Output.ACT.CW.INHIBIT_OPREATION )
   END_RUNG
   RUNG wire#w1
      Contact( #SWITCH_ON )
      Contact( #EMCY_STOP )
      Contact( #Input.ACT.SW.OFF2_STATE )
      Contact( #Input.ACT.SW.OFF3_STATE )
      Contact( #Input.ACT.SW.RDY_ON )
      { S7_GenerateENO := "TRUE" } Move(in := 50, out1 => #POWER_STATE)
   END_RUNG
   // the same network as SCL:
   #_w1 := #POWER_STATE >= 40;
   #Output.ACT.CW.OFF1 := #_w1 AND #START AND #RESTART;
   #Output.ACT.CW.OFF2 := #_w1 AND #SWITCH_ON;
   #Output.ACT.CW.OFF3 := #_w1 AND #EMCY_STOP AND #RESTART_EMG;
   #Output.ACT.CW.INHIBIT_OPREATION := #_w1 AND NOT #COAST_STOP;
   IF #_w1 AND #SWITCH_ON AND #EMCY_STOP AND #Input.ACT.SW.OFF2_STATE AND #Input.ACT.SW.OFF3_STATE AND #Input.ACT.SW.RDY_ON THEN
       #POWER_STATE := 50;
   END_IF;
END_REGION

REGION Network 42: End if not ready to next step
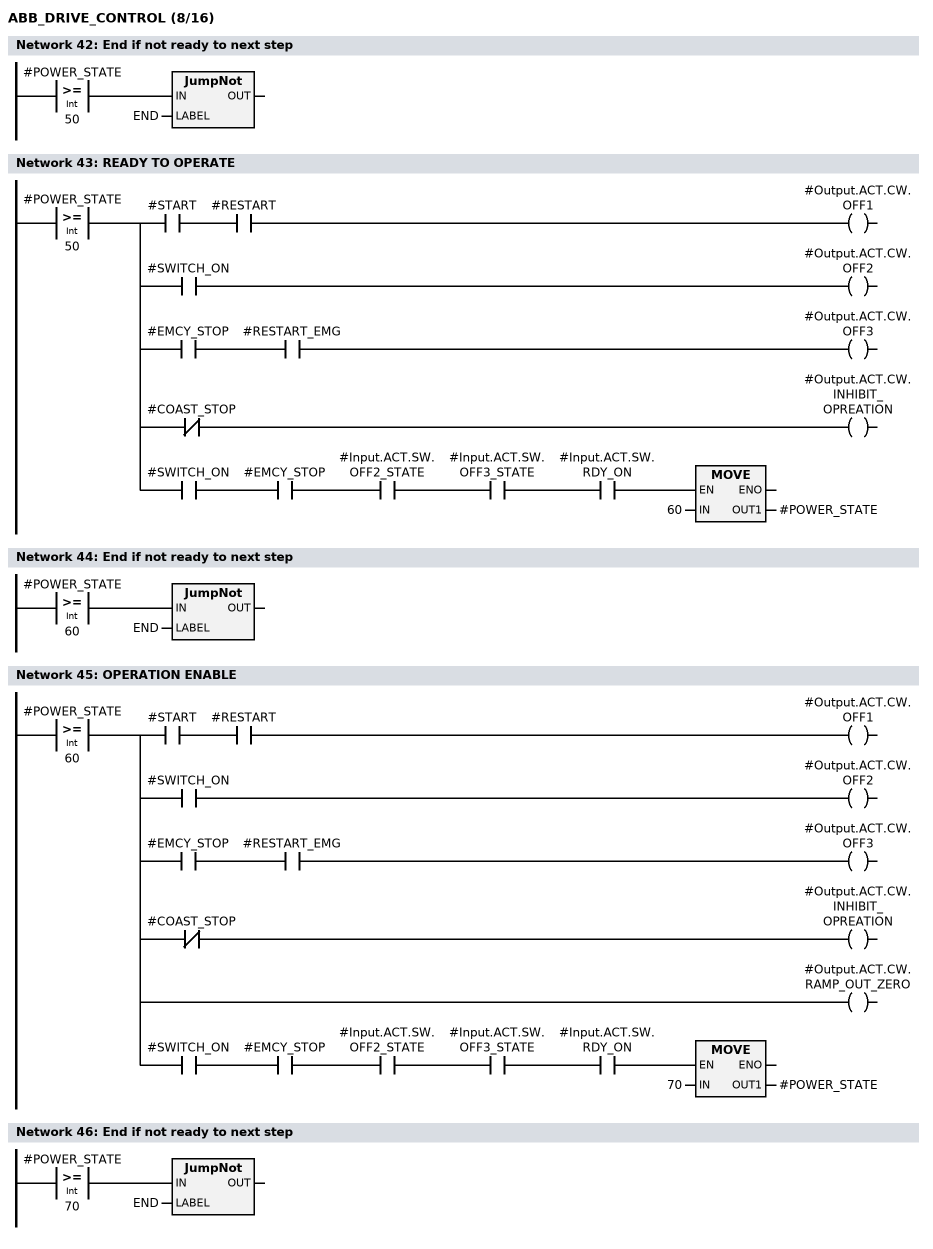
   // no SCL statement known for JumpNot: written as a call
   JumpNot(in := #POWER_STATE >= 50, label := END);
END_REGION

REGION Network 43: READY TO OPERATE
   RUNG wire#powerrail
      { S7_Templates := "SrcType := Int" } GE_Contact(in1 := #POWER_STATE, in2 := 50)
      wire#w1
      Contact( #START )
      Contact( #RESTART )
      Coil( #Output.ACT.CW.OFF1 )
   END_RUNG
   RUNG wire#w1
      Contact( #SWITCH_ON )
      Coil( #Output.ACT.CW.OFF2 )
   END_RUNG
   RUNG wire#w1
      Contact( #EMCY_STOP )
      Contact( #RESTART_EMG )
      Coil( #Output.ACT.CW.OFF3 )
   END_RUNG
   RUNG wire#w1
      I_Contact( #COAST_STOP )
      Coil( #Output.ACT.CW.INHIBIT_OPREATION )
   END_RUNG
   RUNG wire#w1
      Contact( #SWITCH_ON )
      Contact( #EMCY_STOP )
      Contact( #Input.ACT.SW.OFF2_STATE )
      Contact( #Input.ACT.SW.OFF3_STATE )
      Contact( #Input.ACT.SW.RDY_ON )
      { S7_GenerateENO := "TRUE" } Move(in := 60, out1 => #POWER_STATE)
   END_RUNG
   // the same network as SCL:
   #_w1 := #POWER_STATE >= 50;
   #Output.ACT.CW.OFF1 := #_w1 AND #START AND #RESTART;
   #Output.ACT.CW.OFF2 := #_w1 AND #SWITCH_ON;
   #Output.ACT.CW.OFF3 := #_w1 AND #EMCY_STOP AND #RESTART_EMG;
   #Output.ACT.CW.INHIBIT_OPREATION := #_w1 AND NOT #COAST_STOP;
   IF #_w1 AND #SWITCH_ON AND #EMCY_STOP AND #Input.ACT.SW.OFF2_STATE AND #Input.ACT.SW.OFF3_STATE AND #Input.ACT.SW.RDY_ON THEN
       #POWER_STATE := 60;
   END_IF;
END_REGION

REGION Network 44: End if not ready to next step
   // no SCL statement known for JumpNot: written as a call
   JumpNot(in := #POWER_STATE >= 60, label := END);
END_REGION

REGION Network 45: OPERATION ENABLE
   RUNG wire#powerrail
      { S7_Templates := "SrcType := Int" } GE_Contact(in1 := #POWER_STATE, in2 := 60)
      wire#w1
      Contact( #START )
      Contact( #RESTART )
      Coil( #Output.ACT.CW.OFF1 )
   END_RUNG
   RUNG wire#w1
      Contact( #SWITCH_ON )
      Coil( #Output.ACT.CW.OFF2 )
   END_RUNG
   RUNG wire#w1
      Contact( #EMCY_STOP )
      Contact( #RESTART_EMG )
      Coil( #Output.ACT.CW.OFF3 )
   END_RUNG
   RUNG wire#w1
      I_Contact( #COAST_STOP )
      Coil( #Output.ACT.CW.INHIBIT_OPREATION )
   END_RUNG
   RUNG wire#w1
      Coil( #Output.ACT.CW.RAMP_OUT_ZERO )
   END_RUNG
   RUNG wire#w1
      Contact( #SWITCH_ON )
      Contact( #EMCY_STOP )
      Contact( #Input.ACT.SW.OFF2_STATE )
      Contact( #Input.ACT.SW.OFF3_STATE )
      Contact( #Input.ACT.SW.RDY_ON )
      { S7_GenerateENO := "TRUE" } Move(in := 70, out1 => #POWER_STATE)
   END_RUNG
   // the same network as SCL:
   #_w1 := #POWER_STATE >= 60;
   #Output.ACT.CW.OFF1 := #_w1 AND #START AND #RESTART;
   #Output.ACT.CW.OFF2 := #_w1 AND #SWITCH_ON;
   #Output.ACT.CW.OFF3 := #_w1 AND #EMCY_STOP AND #RESTART_EMG;
   #Output.ACT.CW.INHIBIT_OPREATION := #_w1 AND NOT #COAST_STOP;
   #Output.ACT.CW.RAMP_OUT_ZERO := #_w1;
   IF #_w1 AND #SWITCH_ON AND #EMCY_STOP AND #Input.ACT.SW.OFF2_STATE AND #Input.ACT.SW.OFF3_STATE AND #Input.ACT.SW.RDY_ON THEN
       #POWER_STATE := 70;
   END_IF;
END_REGION

REGION Network 46: End if not ready to next step
   // no SCL statement known for JumpNot: written as a call
   JumpNot(in := #POWER_STATE >= 70, label := END);
END_REGION

REGION Network 47: SET RAMP HOLD
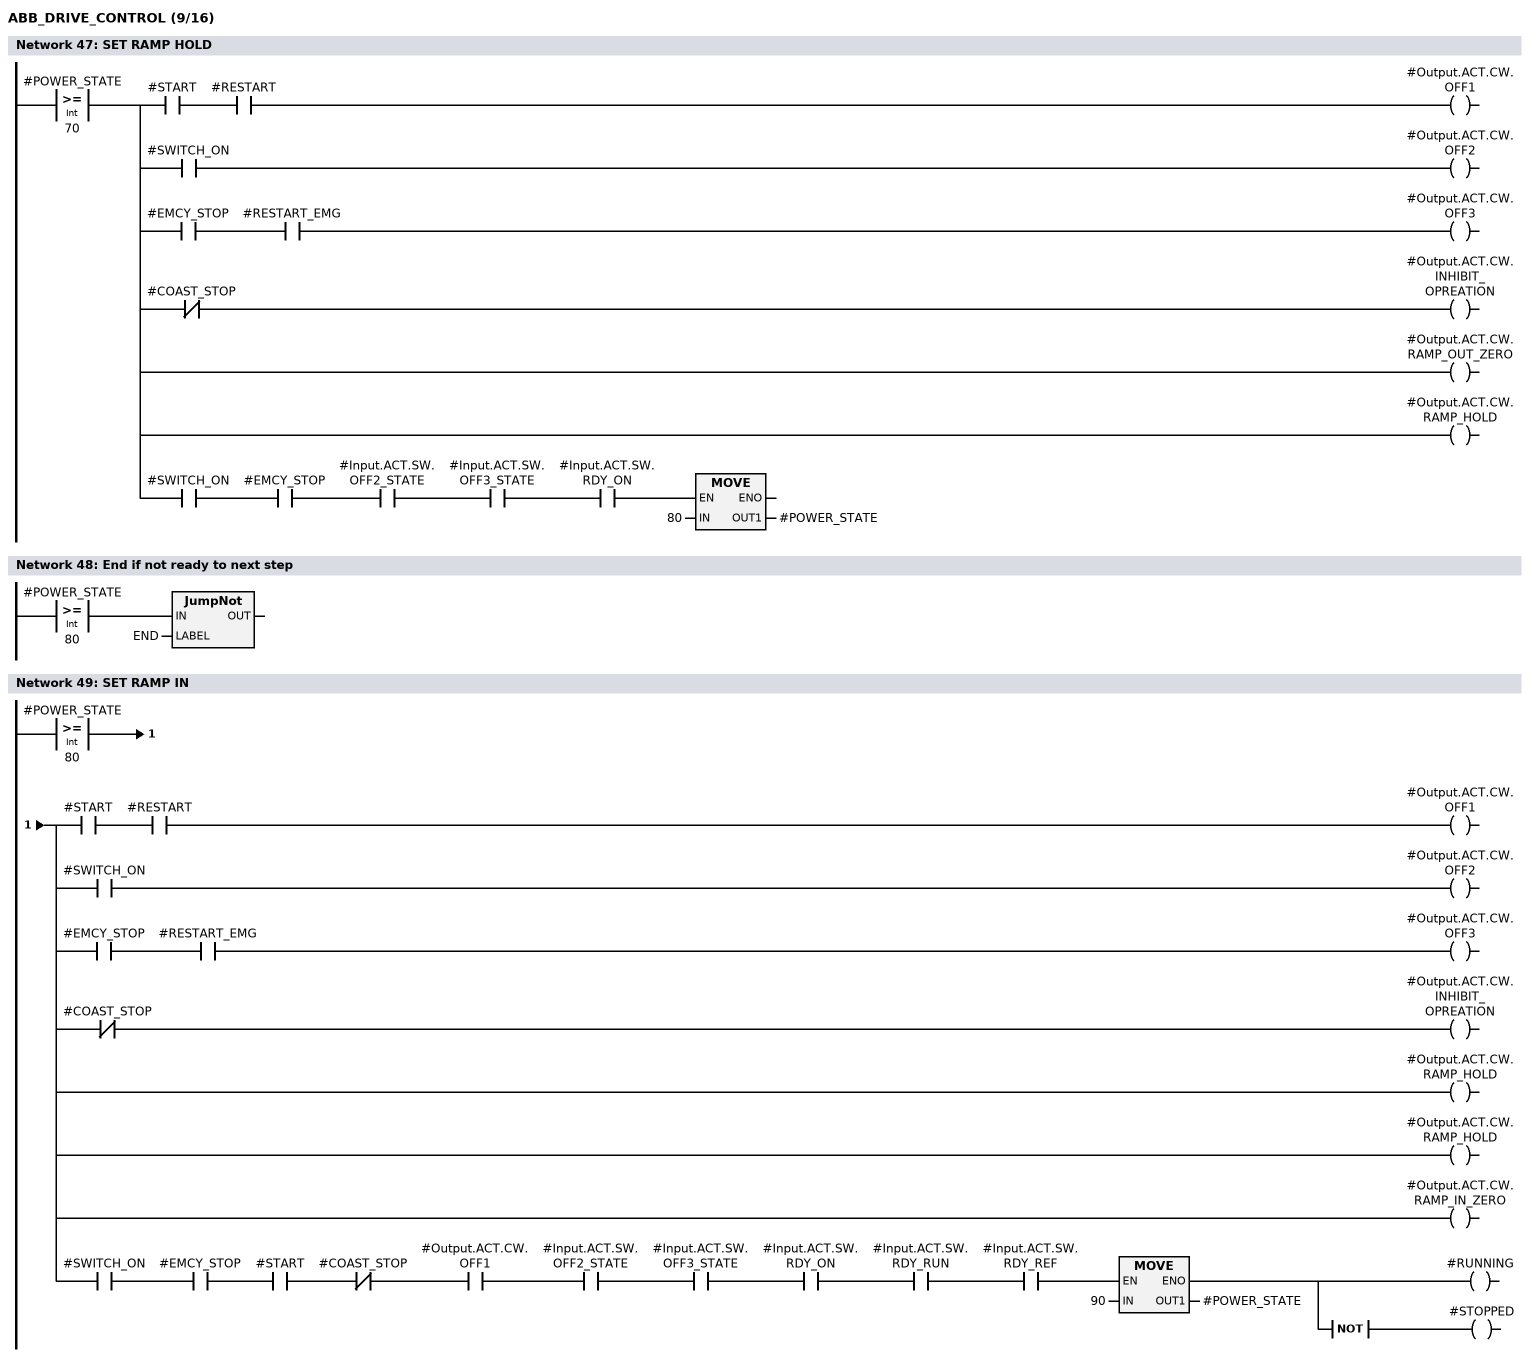
   RUNG wire#powerrail
      { S7_Templates := "SrcType := Int" } GE_Contact(in1 := #POWER_STATE, in2 := 70)
      wire#w1
      Contact( #START )
      Contact( #RESTART )
      Coil( #Output.ACT.CW.OFF1 )
   END_RUNG
   RUNG wire#w1
      Contact( #SWITCH_ON )
      Coil( #Output.ACT.CW.OFF2 )
   END_RUNG
   RUNG wire#w1
      Contact( #EMCY_STOP )
      Contact( #RESTART_EMG )
      Coil( #Output.ACT.CW.OFF3 )
   END_RUNG
   RUNG wire#w1
      I_Contact( #COAST_STOP )
      Coil( #Output.ACT.CW.INHIBIT_OPREATION )
   END_RUNG
   RUNG wire#w1
      Coil( #Output.ACT.CW.RAMP_OUT_ZERO )
   END_RUNG
   RUNG wire#w1
      Coil( #Output.ACT.CW.RAMP_HOLD )
   END_RUNG
   RUNG wire#w1
      Contact( #SWITCH_ON )
      Contact( #EMCY_STOP )
      Contact( #Input.ACT.SW.OFF2_STATE )
      Contact( #Input.ACT.SW.OFF3_STATE )
      Contact( #Input.ACT.SW.RDY_ON )
      { S7_GenerateENO := "TRUE" } Move(in := 80, out1 => #POWER_STATE)
   END_RUNG
   // the same network as SCL:
   #_w1 := #POWER_STATE >= 70;
   #Output.ACT.CW.OFF1 := #_w1 AND #START AND #RESTART;
   #Output.ACT.CW.OFF2 := #_w1 AND #SWITCH_ON;
   #Output.ACT.CW.OFF3 := #_w1 AND #EMCY_STOP AND #RESTART_EMG;
   #Output.ACT.CW.INHIBIT_OPREATION := #_w1 AND NOT #COAST_STOP;
   #Output.ACT.CW.RAMP_OUT_ZERO := #_w1;
   #Output.ACT.CW.RAMP_HOLD := #_w1;
   IF #_w1 AND #SWITCH_ON AND #EMCY_STOP AND #Input.ACT.SW.OFF2_STATE AND #Input.ACT.SW.OFF3_STATE AND #Input.ACT.SW.RDY_ON THEN
       #POWER_STATE := 80;
   END_IF;
END_REGION

REGION Network 48: End if not ready to next step
   // no SCL statement known for JumpNot: written as a call
   JumpNot(in := #POWER_STATE >= 80, label := END);
END_REGION

REGION Network 49: SET RAMP IN
   RUNG wire#powerrail
      { S7_Templates := "SrcType := Int" } GE_Contact(in1 := #POWER_STATE, in2 := 80)
      wire#w1
      Contact( #START )
      Contact( #RESTART )
      Coil( #Output.ACT.CW.OFF1 )
   END_RUNG
   RUNG wire#w1
      Contact( #SWITCH_ON )
      Coil( #Output.ACT.CW.OFF2 )
   END_RUNG
   RUNG wire#w1
      Contact( #EMCY_STOP )
      Contact( #RESTART_EMG )
      Coil( #Output.ACT.CW.OFF3 )
   END_RUNG
   RUNG wire#w1
      I_Contact( #COAST_STOP )
      Coil( #Output.ACT.CW.INHIBIT_OPREATION )
   END_RUNG
   RUNG wire#w1
      Coil( #Output.ACT.CW.RAMP_HOLD )
   END_RUNG
   RUNG wire#w1
      Coil( #Output.ACT.CW.RAMP_HOLD )
   END_RUNG
   RUNG wire#w1
      Coil( #Output.ACT.CW.RAMP_IN_ZERO )
   END_RUNG
   RUNG wire#w1
      Contact( #SWITCH_ON )
      Contact( #EMCY_STOP )
      Contact( #START )
      I_Contact( #COAST_STOP )
      Contact( #Output.ACT.CW.OFF1 )
      Contact( #Input.ACT.SW.OFF2_STATE )
      Contact( #Input.ACT.SW.OFF3_STATE )
      Contact( #Input.ACT.SW.RDY_ON )
      Contact( #Input.ACT.SW.RDY_RUN )
      Contact( #Input.ACT.SW.RDY_REF )
      { S7_GenerateENO := "TRUE" } Move(in := 90, out1 => #POWER_STATE)
      wire#w2
      Coil( #RUNNING )
   END_RUNG
   RUNG wire#w2
      Not()
      Coil( #STOPPED )
   END_RUNG
   // the same network as SCL:
   // ENO of a box is taken as its EN; it also drops when the box reports an error
   #_w1 := #POWER_STATE >= 80;
   #Output.ACT.CW.OFF1 := #_w1 AND #START AND #RESTART;
   #Output.ACT.CW.OFF2 := #_w1 AND #SWITCH_ON;
   #Output.ACT.CW.OFF3 := #_w1 AND #EMCY_STOP AND #RESTART_EMG;
   #Output.ACT.CW.INHIBIT_OPREATION := #_w1 AND NOT #COAST_STOP;
   #Output.ACT.CW.RAMP_HOLD := #_w1;
   #Output.ACT.CW.RAMP_HOLD := #_w1;
   #Output.ACT.CW.RAMP_IN_ZERO := #_w1;
   #_w2 := #_w1 AND #SWITCH_ON AND #EMCY_STOP AND #START AND NOT #COAST_STOP AND #Output.ACT.CW.OFF1 AND #Input.ACT.SW.OFF2_STATE AND #Input.ACT.SW.OFF3_STATE AND #Input.ACT.SW.RDY_ON AND #Input.ACT.SW.RDY_RUN AND #Input.ACT.SW.RDY_REF;
   IF #_w2 THEN #POWER_STATE := 90; END_IF;
   #RUNNING := #_w2;
   #STOPPED := NOT #_w2;
END_REGION

REGION Network 50: End if not ready to next step
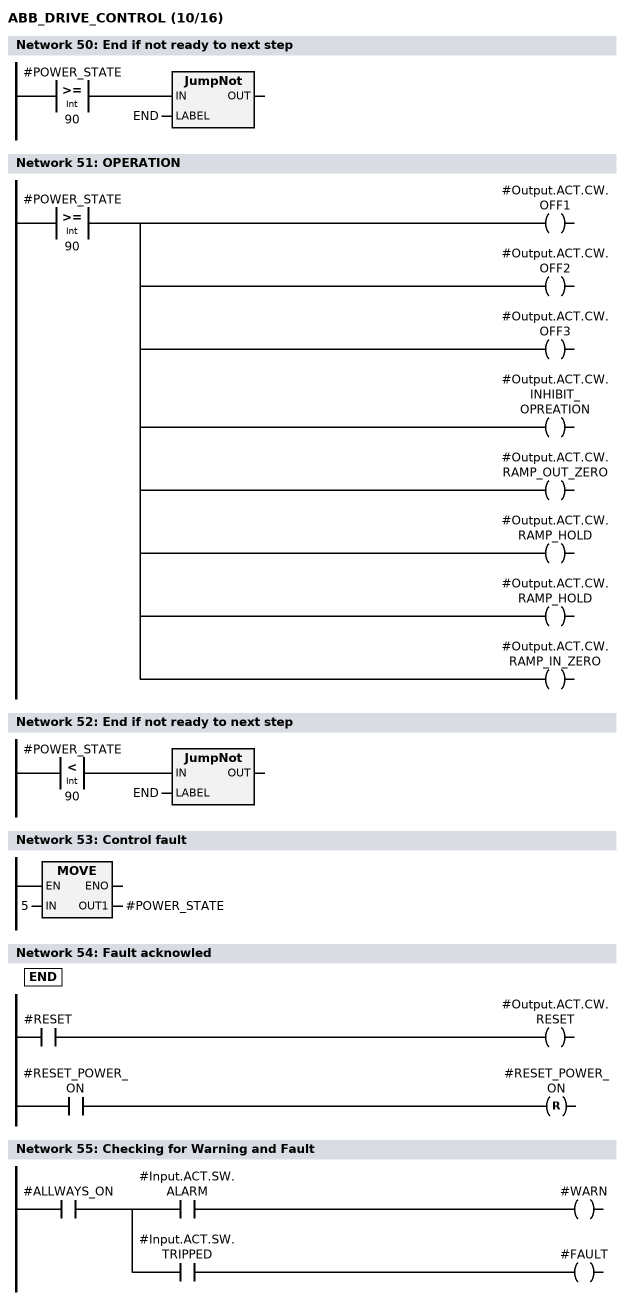
   // no SCL statement known for JumpNot: written as a call
   JumpNot(in := #POWER_STATE >= 90, label := END);
END_REGION

REGION Network 51: OPERATION
   RUNG wire#powerrail
      { S7_Templates := "SrcType := Int" } GE_Contact(in1 := #POWER_STATE, in2 := 90)
      wire#w1
      Coil( #Output.ACT.CW.OFF1 )
   END_RUNG
   RUNG wire#w1
      Coil( #Output.ACT.CW.OFF2 )
   END_RUNG
   RUNG wire#w1
      Coil( #Output.ACT.CW.OFF3 )
   END_RUNG
   RUNG wire#w1
      Coil( #Output.ACT.CW.INHIBIT_OPREATION )
   END_RUNG
   RUNG wire#w1
      Coil( #Output.ACT.CW.RAMP_OUT_ZERO )
   END_RUNG
   RUNG wire#w1
      Coil( #Output.ACT.CW.RAMP_HOLD )
   END_RUNG
   RUNG wire#w1
      Coil( #Output.ACT.CW.RAMP_HOLD )
   END_RUNG
   RUNG wire#w1
      Coil( #Output.ACT.CW.RAMP_IN_ZERO )
   END_RUNG
   // the same network as SCL:
   #Output.ACT.CW.OFF1 := #POWER_STATE >= 90;
   #Output.ACT.CW.OFF2 := #Output.ACT.CW.OFF1;
   #Output.ACT.CW.OFF3 := #Output.ACT.CW.OFF1;
   #Output.ACT.CW.INHIBIT_OPREATION := #Output.ACT.CW.OFF1;
   #Output.ACT.CW.RAMP_OUT_ZERO := #Output.ACT.CW.OFF1;
   #Output.ACT.CW.RAMP_HOLD := #Output.ACT.CW.OFF1;
   #Output.ACT.CW.RAMP_HOLD := #Output.ACT.CW.OFF1;
   #Output.ACT.CW.RAMP_IN_ZERO := #Output.ACT.CW.OFF1;
END_REGION

REGION Network 52: End if not ready to next step
   // no SCL statement known for JumpNot: written as a call
   JumpNot(in := #POWER_STATE < 90, label := END);
END_REGION

REGION Network 53: Control fault
   RUNG wire#powerrail
      { S7_GenerateENO := "TRUE" } Move(in := 5, out1 => #POWER_STATE)
   END_RUNG
   // the same network as SCL:
   #POWER_STATE := 5;
END_REGION

REGION Network 54: Fault acknowled
   Label( END )
   RUNG wire#powerrail
      Contact( #RESET )
      Coil( #Output.ACT.CW.RESET )
   END_RUNG
   RUNG wire#powerrail
      Contact( #RESET_POWER_ON )
      R_Coil( #RESET_POWER_ON )
   END_RUNG
   // the same network as SCL:
   END:
   #Output.ACT.CW.RESET := #RESET;
   IF #RESET_POWER_ON THEN #RESET_POWER_ON := FALSE; END_IF;
END_REGION

REGION Network 55: Checking for Warning and Fault
   RUNG wire#powerrail
      Contact( #ALLWAYS_ON )
      wire#w1
      Contact( #Input.ACT.SW.ALARM )
      Coil( #WARN )
   END_RUNG
   RUNG wire#w1
      Contact( #Input.ACT.SW.TRIPPED )
      Coil( #FAULT )
   END_RUNG
   // the same network as SCL:
   #WARN := #ALLWAYS_ON AND #Input.ACT.SW.ALARM;
   #FAULT := #ALLWAYS_ON AND #Input.ACT.SW.TRIPPED;
END_REGION

REGION Network 56: ReffSpeed
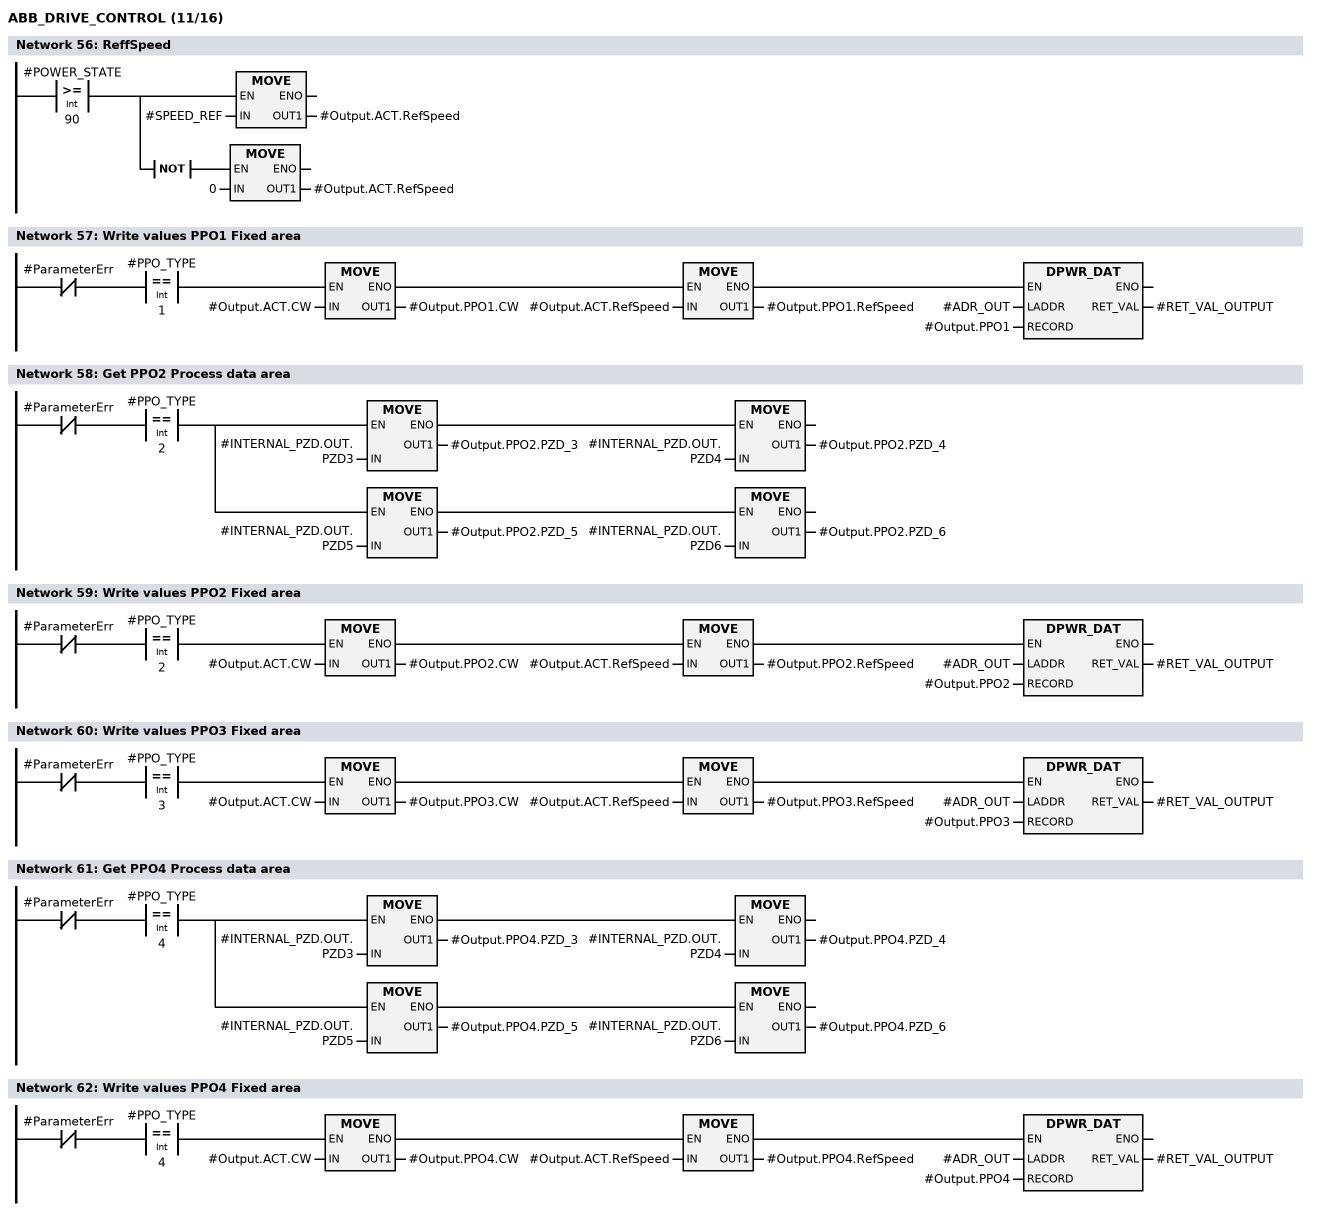
   RUNG wire#powerrail
      { S7_Templates := "SrcType := Int" } GE_Contact(in1 := #POWER_STATE, in2 := 90)
      wire#w1
      { S7_GenerateENO := "TRUE" } Move(in := #SPEED_REF, out1 => #Output.ACT.RefSpeed)
   END_RUNG
   RUNG wire#w1
      Not()
      { S7_GenerateENO := "TRUE" } Move(in := 0, out1 => #Output.ACT.RefSpeed)
   END_RUNG
   // the same network as SCL:
   #_w1 := #POWER_STATE >= 90;
   IF #_w1 THEN #Output.ACT.RefSpeed := #SPEED_REF; END_IF;
   IF NOT #_w1 THEN #Output.ACT.RefSpeed := 0; END_IF;
END_REGION

REGION Network 57: Write values PPO1 Fixed area
   // ENO of a box is taken as its EN; it also drops when the box reports an error
   IF NOT #ParameterErr AND (#PPO_TYPE = 1) THEN
       #Output.PPO1.CW := #Output.ACT.CW;
       #Output.PPO1.RefSpeed := #Output.ACT.RefSpeed;
       #RET_VAL_OUTPUT := DPWR_DAT(LADDR := #ADR_OUT, RECORD := #Output.PPO1);
   END_IF;
END_REGION

REGION Network 58: Get PPO2 Process data area
   RUNG wire#powerrail
      I_Contact( #ParameterErr )
      { S7_Templates := "SrcType := Int" } EQ_Contact(in1 := #PPO_TYPE, in2 := 2)
      wire#w1
      { S7_GenerateENO := "TRUE" } Move(in := #INTERNAL_PZD.OUT.PZD3, out1 => #Output.PPO2.PZD_3)
      { S7_GenerateENO := "TRUE" } Move(in := #INTERNAL_PZD.OUT.PZD4, out1 => #Output.PPO2.PZD_4)
   END_RUNG
   RUNG wire#w1
      { S7_GenerateENO := "TRUE" } Move(in := #INTERNAL_PZD.OUT.PZD5, out1 => #Output.PPO2.PZD_5)
      { S7_GenerateENO := "TRUE" } Move(in := #INTERNAL_PZD.OUT.PZD6, out1 => #Output.PPO2.PZD_6)
   END_RUNG
   // the same network as SCL:
   // ENO of a box is taken as its EN; it also drops when the box reports an error
   IF NOT #ParameterErr AND (#PPO_TYPE = 2) THEN
       #Output.PPO2.PZD_3 := #INTERNAL_PZD.OUT.PZD3;
       #Output.PPO2.PZD_4 := #INTERNAL_PZD.OUT.PZD4;
       #Output.PPO2.PZD_5 := #INTERNAL_PZD.OUT.PZD5;
       #Output.PPO2.PZD_6 := #INTERNAL_PZD.OUT.PZD6;
   END_IF;
END_REGION

REGION Network 59: Write values PPO2 Fixed area
   // ENO of a box is taken as its EN; it also drops when the box reports an error
   IF NOT #ParameterErr AND (#PPO_TYPE = 2) THEN
       #Output.PPO2.CW := #Output.ACT.CW;
       #Output.PPO2.RefSpeed := #Output.ACT.RefSpeed;
       #RET_VAL_OUTPUT := DPWR_DAT(LADDR := #ADR_OUT, RECORD := #Output.PPO2);
   END_IF;
END_REGION

REGION Network 60: Write values PPO3 Fixed area
   // ENO of a box is taken as its EN; it also drops when the box reports an error
   IF NOT #ParameterErr AND (#PPO_TYPE = 3) THEN
       #Output.PPO3.CW := #Output.ACT.CW;
       #Output.PPO3.RefSpeed := #Output.ACT.RefSpeed;
       #RET_VAL_OUTPUT := DPWR_DAT(LADDR := #ADR_OUT, RECORD := #Output.PPO3);
   END_IF;
END_REGION

REGION Network 61: Get PPO4 Process data area
   RUNG wire#powerrail
      I_Contact( #ParameterErr )
      { S7_Templates := "SrcType := Int" } EQ_Contact(in1 := #PPO_TYPE, in2 := 4)
      wire#w1
      { S7_GenerateENO := "TRUE" } Move(in := #INTERNAL_PZD.OUT.PZD3, out1 => #Output.PPO4.PZD_3)
      { S7_GenerateENO := "TRUE" } Move(in := #INTERNAL_PZD.OUT.PZD4, out1 => #Output.PPO4.PZD_4)
   END_RUNG
   RUNG wire#w1
      { S7_GenerateENO := "TRUE" } Move(in := #INTERNAL_PZD.OUT.PZD5, out1 => #Output.PPO4.PZD_5)
      { S7_GenerateENO := "TRUE" } Move(in := #INTERNAL_PZD.OUT.PZD6, out1 => #Output.PPO4.PZD_6)
   END_RUNG
   // the same network as SCL:
   // ENO of a box is taken as its EN; it also drops when the box reports an error
   IF NOT #ParameterErr AND (#PPO_TYPE = 4) THEN
       #Output.PPO4.PZD_3 := #INTERNAL_PZD.OUT.PZD3;
       #Output.PPO4.PZD_4 := #INTERNAL_PZD.OUT.PZD4;
       #Output.PPO4.PZD_5 := #INTERNAL_PZD.OUT.PZD5;
       #Output.PPO4.PZD_6 := #INTERNAL_PZD.OUT.PZD6;
   END_IF;
END_REGION

REGION Network 62: Write values PPO4 Fixed area
   // ENO of a box is taken as its EN; it also drops when the box reports an error
   IF NOT #ParameterErr AND (#PPO_TYPE = 4) THEN
       #Output.PPO4.CW := #Output.ACT.CW;
       #Output.PPO4.RefSpeed := #Output.ACT.RefSpeed;
       #RET_VAL_OUTPUT := DPWR_DAT(LADDR := #ADR_OUT, RECORD := #Output.PPO4);
   END_IF;
END_REGION

REGION Network 63: Get PPO5 Process data area
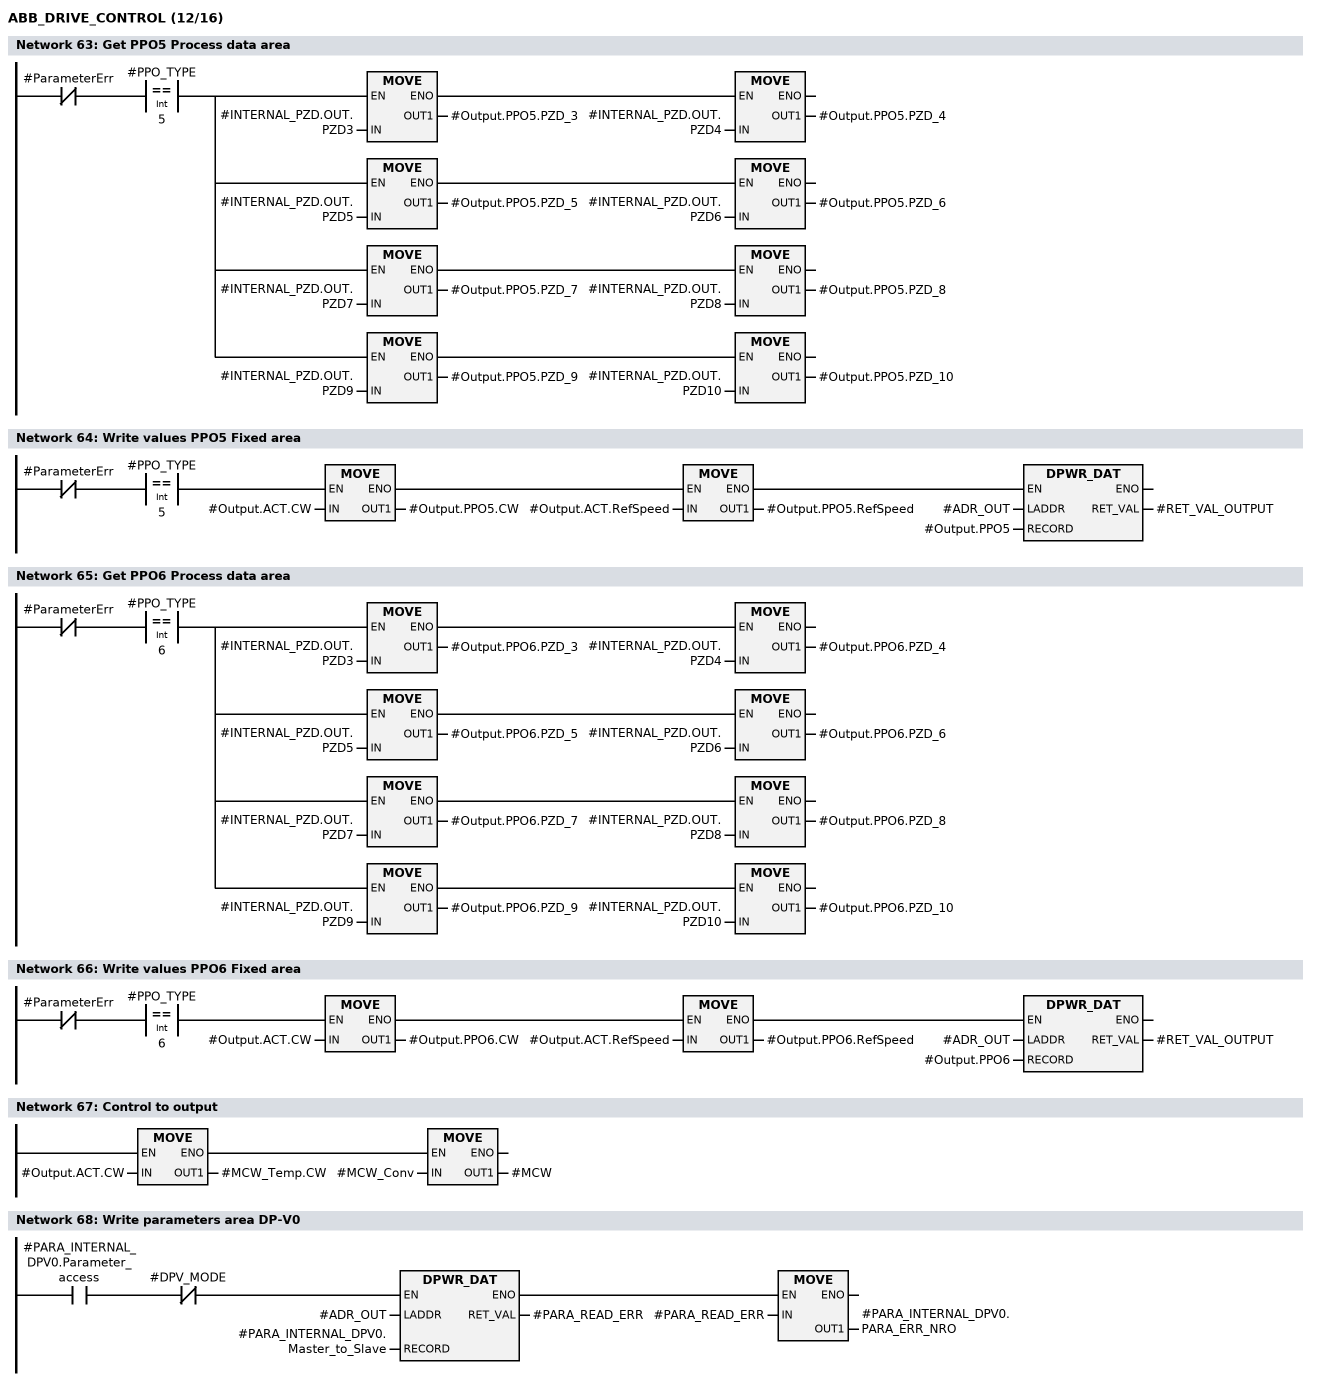
   RUNG wire#powerrail
      I_Contact( #ParameterErr )
      { S7_Templates := "SrcType := Int" } EQ_Contact(in1 := #PPO_TYPE, in2 := 5)
      wire#w1
      { S7_GenerateENO := "TRUE" } Move(in := #INTERNAL_PZD.OUT.PZD3, out1 => #Output.PPO5.PZD_3)
      { S7_GenerateENO := "TRUE" } Move(in := #INTERNAL_PZD.OUT.PZD4, out1 => #Output.PPO5.PZD_4)
   END_RUNG
   RUNG wire#w1
      { S7_GenerateENO := "TRUE" } Move(in := #INTERNAL_PZD.OUT.PZD5, out1 => #Output.PPO5.PZD_5)
      { S7_GenerateENO := "TRUE" } Move(in := #INTERNAL_PZD.OUT.PZD6, out1 => #Output.PPO5.PZD_6)
   END_RUNG
   RUNG wire#w1
      { S7_GenerateENO := "TRUE" } Move(in := #INTERNAL_PZD.OUT.PZD7, out1 => #Output.PPO5.PZD_7)
      { S7_GenerateENO := "TRUE" } Move(in := #INTERNAL_PZD.OUT.PZD8, out1 => #Output.PPO5.PZD_8)
   END_RUNG
   RUNG wire#w1
      { S7_GenerateENO := "TRUE" } Move(in := #INTERNAL_PZD.OUT.PZD9, out1 => #Output.PPO5.PZD_9)
      { S7_GenerateENO := "TRUE" } Move(in := #INTERNAL_PZD.OUT.PZD10, out1 => #Output.PPO5.PZD_10)
   END_RUNG
   // the same network as SCL:
   // ENO of a box is taken as its EN; it also drops when the box reports an error
   IF NOT #ParameterErr AND (#PPO_TYPE = 5) THEN
       #Output.PPO5.PZD_3 := #INTERNAL_PZD.OUT.PZD3;
       #Output.PPO5.PZD_4 := #INTERNAL_PZD.OUT.PZD4;
       #Output.PPO5.PZD_5 := #INTERNAL_PZD.OUT.PZD5;
       #Output.PPO5.PZD_6 := #INTERNAL_PZD.OUT.PZD6;
       #Output.PPO5.PZD_7 := #INTERNAL_PZD.OUT.PZD7;
       #Output.PPO5.PZD_8 := #INTERNAL_PZD.OUT.PZD8;
       #Output.PPO5.PZD_9 := #INTERNAL_PZD.OUT.PZD9;
       #Output.PPO5.PZD_10 := #INTERNAL_PZD.OUT.PZD10;
   END_IF;
END_REGION

REGION Network 64: Write values PPO5 Fixed area
   // ENO of a box is taken as its EN; it also drops when the box reports an error
   IF NOT #ParameterErr AND (#PPO_TYPE = 5) THEN
       #Output.PPO5.CW := #Output.ACT.CW;
       #Output.PPO5.RefSpeed := #Output.ACT.RefSpeed;
       #RET_VAL_OUTPUT := DPWR_DAT(LADDR := #ADR_OUT, RECORD := #Output.PPO5);
   END_IF;
END_REGION

REGION Network 65: Get PPO6 Process data area
   RUNG wire#powerrail
      I_Contact( #ParameterErr )
      { S7_Templates := "SrcType := Int" } EQ_Contact(in1 := #PPO_TYPE, in2 := 6)
      wire#w1
      { S7_GenerateENO := "TRUE" } Move(in := #INTERNAL_PZD.OUT.PZD3, out1 => #Output.PPO6.PZD_3)
      { S7_GenerateENO := "TRUE" } Move(in := #INTERNAL_PZD.OUT.PZD4, out1 => #Output.PPO6.PZD_4)
   END_RUNG
   RUNG wire#w1
      { S7_GenerateENO := "TRUE" } Move(in := #INTERNAL_PZD.OUT.PZD5, out1 => #Output.PPO6.PZD_5)
      { S7_GenerateENO := "TRUE" } Move(in := #INTERNAL_PZD.OUT.PZD6, out1 => #Output.PPO6.PZD_6)
   END_RUNG
   RUNG wire#w1
      { S7_GenerateENO := "TRUE" } Move(in := #INTERNAL_PZD.OUT.PZD7, out1 => #Output.PPO6.PZD_7)
      { S7_GenerateENO := "TRUE" } Move(in := #INTERNAL_PZD.OUT.PZD8, out1 => #Output.PPO6.PZD_8)
   END_RUNG
   RUNG wire#w1
      { S7_GenerateENO := "TRUE" } Move(in := #INTERNAL_PZD.OUT.PZD9, out1 => #Output.PPO6.PZD_9)
      { S7_GenerateENO := "TRUE" } Move(in := #INTERNAL_PZD.OUT.PZD10, out1 => #Output.PPO6.PZD_10)
   END_RUNG
   // the same network as SCL:
   // ENO of a box is taken as its EN; it also drops when the box reports an error
   IF NOT #ParameterErr AND (#PPO_TYPE = 6) THEN
       #Output.PPO6.PZD_3 := #INTERNAL_PZD.OUT.PZD3;
       #Output.PPO6.PZD_4 := #INTERNAL_PZD.OUT.PZD4;
       #Output.PPO6.PZD_5 := #INTERNAL_PZD.OUT.PZD5;
       #Output.PPO6.PZD_6 := #INTERNAL_PZD.OUT.PZD6;
       #Output.PPO6.PZD_7 := #INTERNAL_PZD.OUT.PZD7;
       #Output.PPO6.PZD_8 := #INTERNAL_PZD.OUT.PZD8;
       #Output.PPO6.PZD_9 := #INTERNAL_PZD.OUT.PZD9;
       #Output.PPO6.PZD_10 := #INTERNAL_PZD.OUT.PZD10;
   END_IF;
END_REGION

REGION Network 66: Write values PPO6 Fixed area
   // ENO of a box is taken as its EN; it also drops when the box reports an error
   IF NOT #ParameterErr AND (#PPO_TYPE = 6) THEN
       #Output.PPO6.CW := #Output.ACT.CW;
       #Output.PPO6.RefSpeed := #Output.ACT.RefSpeed;
       #RET_VAL_OUTPUT := DPWR_DAT(LADDR := #ADR_OUT, RECORD := #Output.PPO6);
   END_IF;
END_REGION

REGION Network 67: Control to output
   RUNG wire#powerrail
      { S7_GenerateENO := "TRUE" } Move(in := #Output.ACT.CW, out1 => #MCW_Temp.CW)
      { S7_GenerateENO := "TRUE" } Move(in := #MCW_Conv, out1 => #MCW)
   END_RUNG
   // the same network as SCL:
   // ENO of a box is taken as its EN; it also drops when the box reports an error
   #MCW_Temp.CW := #Output.ACT.CW;
   #MCW := #MCW_Conv;
END_REGION

REGION Network 68: Write parameters area DP-V0
   // ENO of a box is taken as its EN; it also drops when the box reports an error
   IF #PARA_INTERNAL_DPV0.Parameter_access AND NOT #DPV_MODE THEN
       #PARA_READ_ERR := DPWR_DAT(LADDR := #ADR_OUT, RECORD := #PARA_INTERNAL_DPV0.Master_to_Slave);
       #PARA_INTERNAL_DPV0.PARA_ERR_NRO := #PARA_READ_ERR;
   END_IF;
END_REGION

REGION Network 69: Error occured during execution when output ERR=TRUE
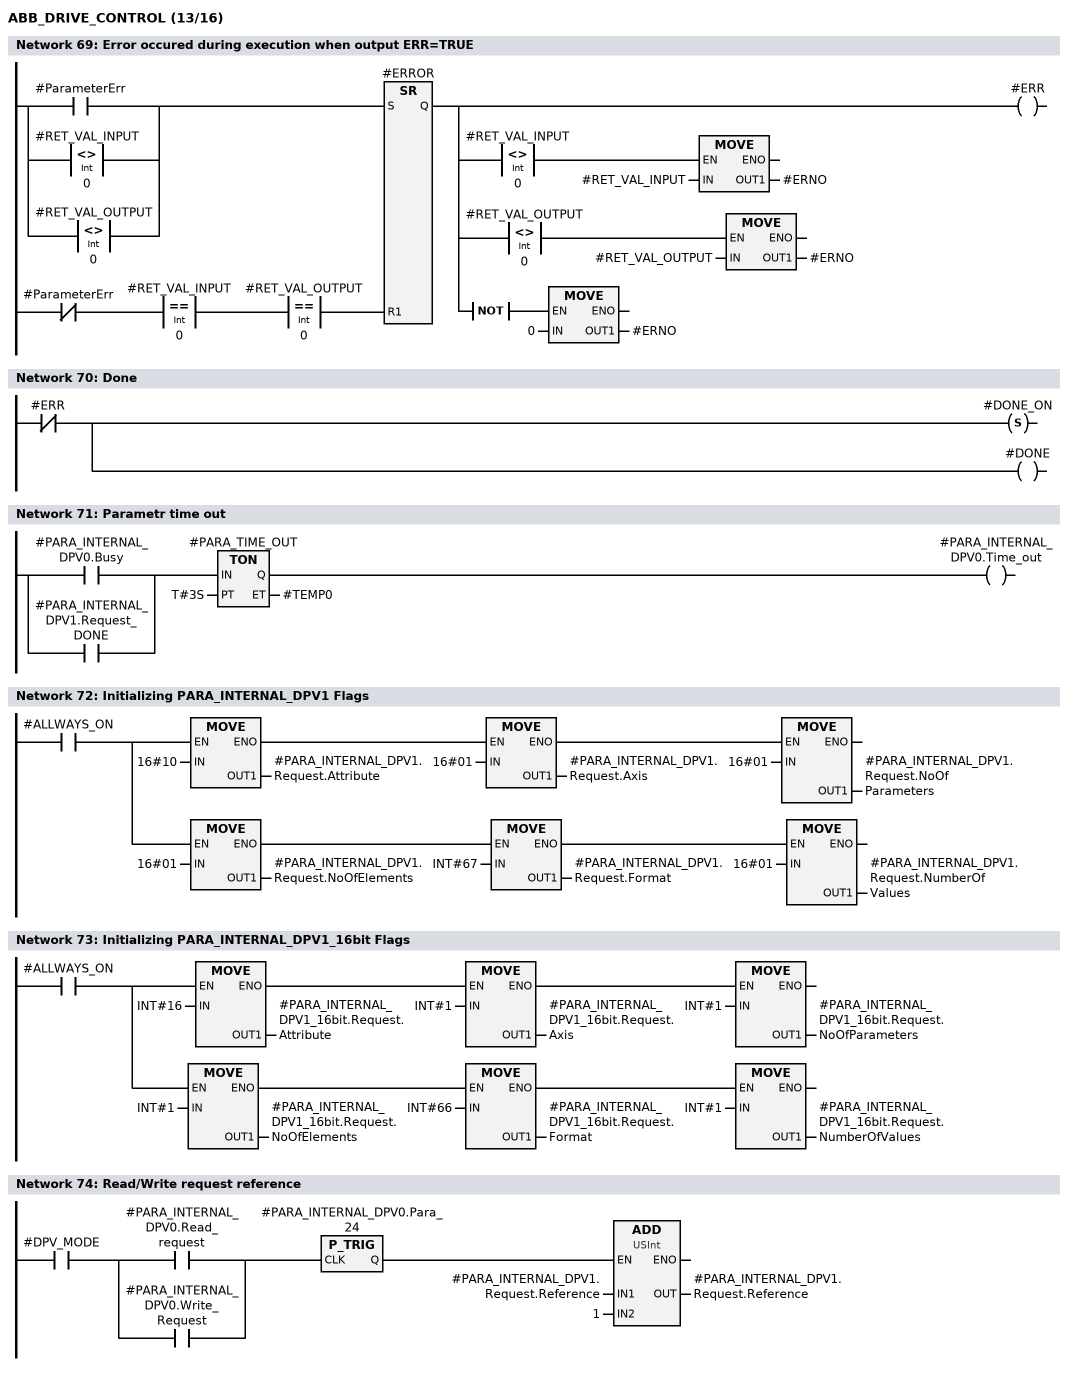
   RUNG wire#powerrail
      Contact( #ParameterErr )
      wire#w1
      S_SR(operand := #ERROR, r1 := wire#w2)
      wire#w3
      Coil( #ERR )
   END_RUNG
   RUNG wire#powerrail
      { S7_Templates := "SrcType := Int" } NE_Contact(in1 := #RET_VAL_INPUT, in2 := 0)
   END_RUNG wire#w1
   RUNG wire#powerrail
      { S7_Templates := "SrcType := Int" } NE_Contact(in1 := #RET_VAL_OUTPUT, in2 := 0)
   END_RUNG wire#w1
   RUNG wire#powerrail
      I_Contact( #ParameterErr )
      { S7_Templates := "SrcType := Int" } EQ_Contact(in1 := #RET_VAL_INPUT, in2 := 0)
      { S7_Templates := "SrcType := Int" } EQ_Contact(in1 := #RET_VAL_OUTPUT, in2 := 0)
   END_RUNG wire#w2
   RUNG wire#w3
      { S7_Templates := "SrcType := Int" } NE_Contact(in1 := #RET_VAL_INPUT, in2 := 0)
      { S7_GenerateENO := "TRUE" } Move(in := #RET_VAL_INPUT, out1 => #ERNO)
   END_RUNG
   RUNG wire#w3
      { S7_Templates := "SrcType := Int" } NE_Contact(in1 := #RET_VAL_OUTPUT, in2 := 0)
      { S7_GenerateENO := "TRUE" } Move(in := #RET_VAL_OUTPUT, out1 => #ERNO)
   END_RUNG
   RUNG wire#w3
      Not()
      { S7_GenerateENO := "TRUE" } Move(in := 0, out1 => #ERNO)
   END_RUNG
   // the same network as SCL:
   IF #ParameterErr OR (#RET_VAL_INPUT <> 0) OR (#RET_VAL_OUTPUT <> 0) THEN
       #ERROR := TRUE;   // SR flip-flop
   END_IF;
   IF NOT #ParameterErr AND (#RET_VAL_INPUT = 0) AND (#RET_VAL_OUTPUT = 0) THEN #ERROR := FALSE; END_IF;
   #ERR := #ERROR;
   IF #ERROR AND (#RET_VAL_INPUT <> 0) THEN #ERNO := #RET_VAL_INPUT; END_IF;
   IF #ERROR AND (#RET_VAL_OUTPUT <> 0) THEN #ERNO := #RET_VAL_OUTPUT; END_IF;
   IF NOT #ERROR THEN #ERNO := 0; END_IF;
END_REGION

REGION Network 70: Done
   RUNG wire#powerrail
      I_Contact( #ERR )
      wire#w1
      S_Coil( #DONE_ON )
   END_RUNG
   RUNG wire#w1
      Coil( #DONE )
   END_RUNG
   // the same network as SCL:
   IF NOT #ERR THEN #DONE_ON := TRUE; END_IF;
   #DONE := NOT #ERR;
END_REGION

REGION Network 71: Parametr time out
   #PARA_TIME_OUT(IN := #PARA_INTERNAL_DPV0.Busy OR #PARA_INTERNAL_DPV1.Request_DONE, PT := T#3S, ET => #TEMP0);   // TON
   #PARA_INTERNAL_DPV0.Time_out := #PARA_TIME_OUT.Q;
END_REGION

REGION Network 72: Initializing PARA_INTERNAL_DPV1 Flags
   RUNG wire#powerrail
      Contact( #ALLWAYS_ON )
      wire#w1
      { S7_GenerateENO := "TRUE" } Move(in := 16#10, out1 => #PARA_INTERNAL_DPV1.Request.Attribute)
      { S7_GenerateENO := "TRUE" } Move(in := 16#01, out1 => #PARA_INTERNAL_DPV1.Request.Axis)
      { S7_GenerateENO := "TRUE" } Move(in := 16#01, out1 => #PARA_INTERNAL_DPV1.Request.NoOfParameters)
   END_RUNG
   RUNG wire#w1
      { S7_GenerateENO := "TRUE" } Move(in := 16#01, out1 => #PARA_INTERNAL_DPV1.Request.NoOfElements)
      { S7_GenerateENO := "TRUE" } Move(in := INT#67, out1 => #PARA_INTERNAL_DPV1.Request.Format)
      { S7_GenerateENO := "TRUE" } Move(in := 16#01, out1 => #PARA_INTERNAL_DPV1.Request.NumberOfValues)
   END_RUNG
   // the same network as SCL:
   // ENO of a box is taken as its EN; it also drops when the box reports an error
   IF #ALLWAYS_ON THEN
       #PARA_INTERNAL_DPV1.Request.Attribute := 16#10;
       #PARA_INTERNAL_DPV1.Request.Axis := 16#01;
       #PARA_INTERNAL_DPV1.Request.NoOfParameters := 16#01;
       #PARA_INTERNAL_DPV1.Request.NoOfElements := 16#01;
       #PARA_INTERNAL_DPV1.Request.Format := INT#67;
       #PARA_INTERNAL_DPV1.Request.NumberOfValues := 16#01;
   END_IF;
END_REGION

REGION Network 73: Initializing PARA_INTERNAL_DPV1_16bit Flags
   RUNG wire#powerrail
      Contact( #ALLWAYS_ON )
      wire#w1
      { S7_GenerateENO := "TRUE" } Move(in := INT#16, out1 => #PARA_INTERNAL_DPV1_16bit.Request.Attribute)
      { S7_GenerateENO := "TRUE" } Move(in := INT#1, out1 => #PARA_INTERNAL_DPV1_16bit.Request.Axis)
      { S7_GenerateENO := "TRUE" } Move(in := INT#1, out1 => #PARA_INTERNAL_DPV1_16bit.Request.NoOfParameters)
   END_RUNG
   RUNG wire#w1
      { S7_GenerateENO := "TRUE" } Move(in := INT#1, out1 => #PARA_INTERNAL_DPV1_16bit.Request.NoOfElements)
      { S7_GenerateENO := "TRUE" } Move(in := INT#66, out1 => #PARA_INTERNAL_DPV1_16bit.Request.Format)
      { S7_GenerateENO := "TRUE" } Move(in := INT#1, out1 => #PARA_INTERNAL_DPV1_16bit.Request.NumberOfValues)
   END_RUNG
   // the same network as SCL:
   // ENO of a box is taken as its EN; it also drops when the box reports an error
   IF #ALLWAYS_ON THEN
       #PARA_INTERNAL_DPV1_16bit.Request.Attribute := INT#16;
       #PARA_INTERNAL_DPV1_16bit.Request.Axis := INT#1;
       #PARA_INTERNAL_DPV1_16bit.Request.NoOfParameters := INT#1;
       #PARA_INTERNAL_DPV1_16bit.Request.NoOfElements := INT#1;
       #PARA_INTERNAL_DPV1_16bit.Request.Format := INT#66;
       #PARA_INTERNAL_DPV1_16bit.Request.NumberOfValues := INT#1;
   END_IF;
END_REGION

REGION Network 74: Read/Write request reference
   RUNG wire#powerrail
      Contact( #DPV_MODE )
      wire#w1
      Contact( #PARA_INTERNAL_DPV0.Read_request )
      wire#w2
      P_Trig( #PARA_INTERNAL_DPV0.Para_24 )
      { S7_Templates := "SrcType := USInt"; S7_GenerateENO := "TRUE" } Add(in1 := #PARA_INTERNAL_DPV1.Request.Reference, in2 := 1, out => #PARA_INTERNAL_DPV1.Request.Reference)
   END_RUNG
   RUNG wire#w1
      Contact( #PARA_INTERNAL_DPV0.Write_Request )
   END_RUNG wire#w2
   // the same network as SCL:
   #_w1 := #DPV_MODE AND (#PARA_INTERNAL_DPV0.Read_request OR #PARA_INTERNAL_DPV0.Write_Request);
   #_w2 := #_w1 AND NOT #PARA_INTERNAL_DPV0.Para_24;   // rising edge
   #PARA_INTERNAL_DPV0.Para_24 := #_w1;
   IF #_w2 THEN #PARA_INTERNAL_DPV1.Request.Reference := #PARA_INTERNAL_DPV1.Request.Reference + 1; END_IF;
END_REGION

REGION Network 75: Read parameter area DP-V1
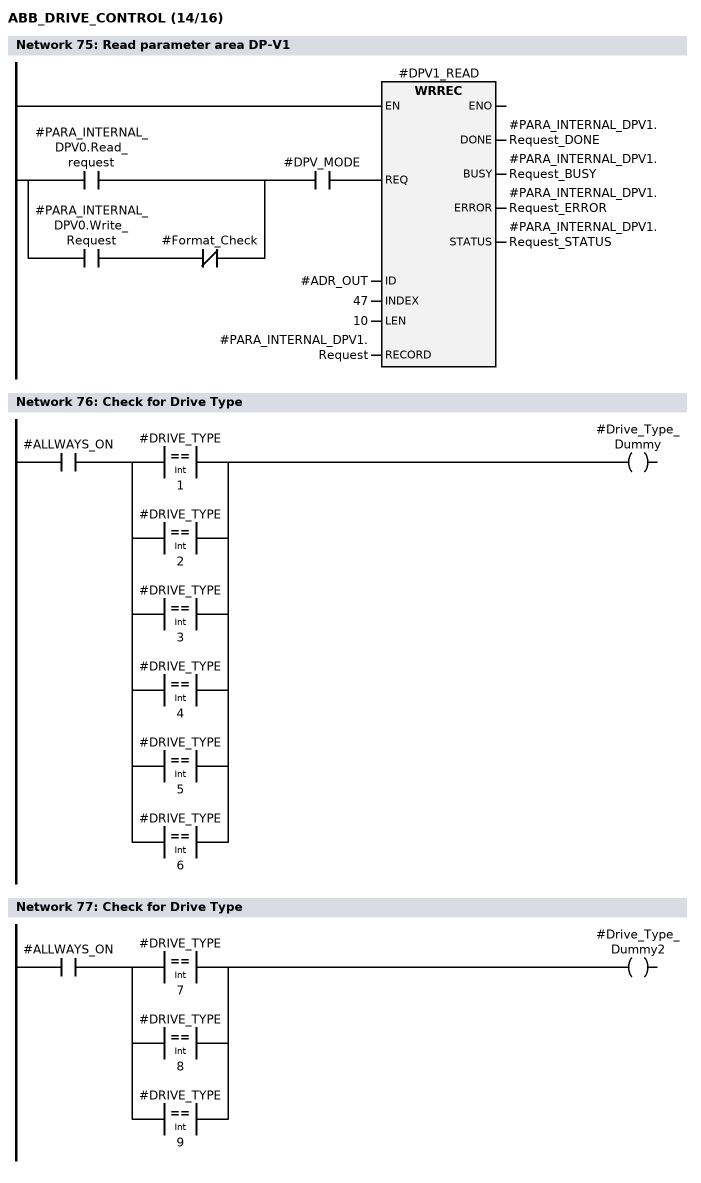
   #DPV1_READ(REQ := (#PARA_INTERNAL_DPV0.Read_request OR (#PARA_INTERNAL_DPV0.Write_Request AND NOT #Format_Check)) AND #DPV_MODE,   // WRREC
              ID := #ADR_OUT,
              INDEX := 47,
              LEN := 10,
              RECORD := #PARA_INTERNAL_DPV1.Request,
              DONE => #PARA_INTERNAL_DPV1.Request_DONE,
              BUSY => #PARA_INTERNAL_DPV1.Request_BUSY,
              ERROR => #PARA_INTERNAL_DPV1.Request_ERROR,
              STATUS => #PARA_INTERNAL_DPV1.Request_STATUS);
END_REGION

REGION Network 76: Check for Drive Type
   RUNG wire#powerrail
      Contact( #ALLWAYS_ON )
      wire#w1
      { S7_Templates := "SrcType := Int" } EQ_Contact(in1 := #DRIVE_TYPE, in2 := 1)
      wire#w2
      Coil( #Drive_Type_Dummy )
   END_RUNG
   RUNG wire#w1
      { S7_Templates := "SrcType := Int" } EQ_Contact(in1 := #DRIVE_TYPE, in2 := 2)
   END_RUNG wire#w2
   RUNG wire#w1
      { S7_Templates := "SrcType := Int" } EQ_Contact(in1 := #DRIVE_TYPE, in2 := 3)
   END_RUNG wire#w2
   RUNG wire#w1
      { S7_Templates := "SrcType := Int" } EQ_Contact(in1 := #DRIVE_TYPE, in2 := 4)
   END_RUNG wire#w2
   RUNG wire#w1
      { S7_Templates := "SrcType := Int" } EQ_Contact(in1 := #DRIVE_TYPE, in2 := 5)
   END_RUNG wire#w2
   RUNG wire#w1
      { S7_Templates := "SrcType := Int" } EQ_Contact(in1 := #DRIVE_TYPE, in2 := 6)
   END_RUNG wire#w2
   // the same network as SCL:
   #Drive_Type_Dummy := #ALLWAYS_ON AND ((#DRIVE_TYPE = 1) OR (#DRIVE_TYPE = 2) OR (#DRIVE_TYPE = 3) OR (#DRIVE_TYPE = 4) OR (#DRIVE_TYPE = 5) OR (#DRIVE_TYPE = 6));
END_REGION

REGION Network 77: Check for Drive Type
   RUNG wire#powerrail
      Contact( #ALLWAYS_ON )
      wire#w1
      { S7_Templates := "SrcType := Int" } EQ_Contact(in1 := #DRIVE_TYPE, in2 := 7)
      wire#w2
      Coil( #Drive_Type_Dummy2 )
   END_RUNG
   RUNG wire#w1
      { S7_Templates := "SrcType := Int" } EQ_Contact(in1 := #DRIVE_TYPE, in2 := 8)
   END_RUNG wire#w2
   RUNG wire#w1
      { S7_Templates := "SrcType := Int" } EQ_Contact(in1 := #DRIVE_TYPE, in2 := 9)
   END_RUNG wire#w2
   // the same network as SCL:
   #Drive_Type_Dummy2 := #ALLWAYS_ON AND ((#DRIVE_TYPE = 7) OR (#DRIVE_TYPE = 8) OR (#DRIVE_TYPE = 9));
END_REGION

REGION Network 78: Check for Parameter Format Type
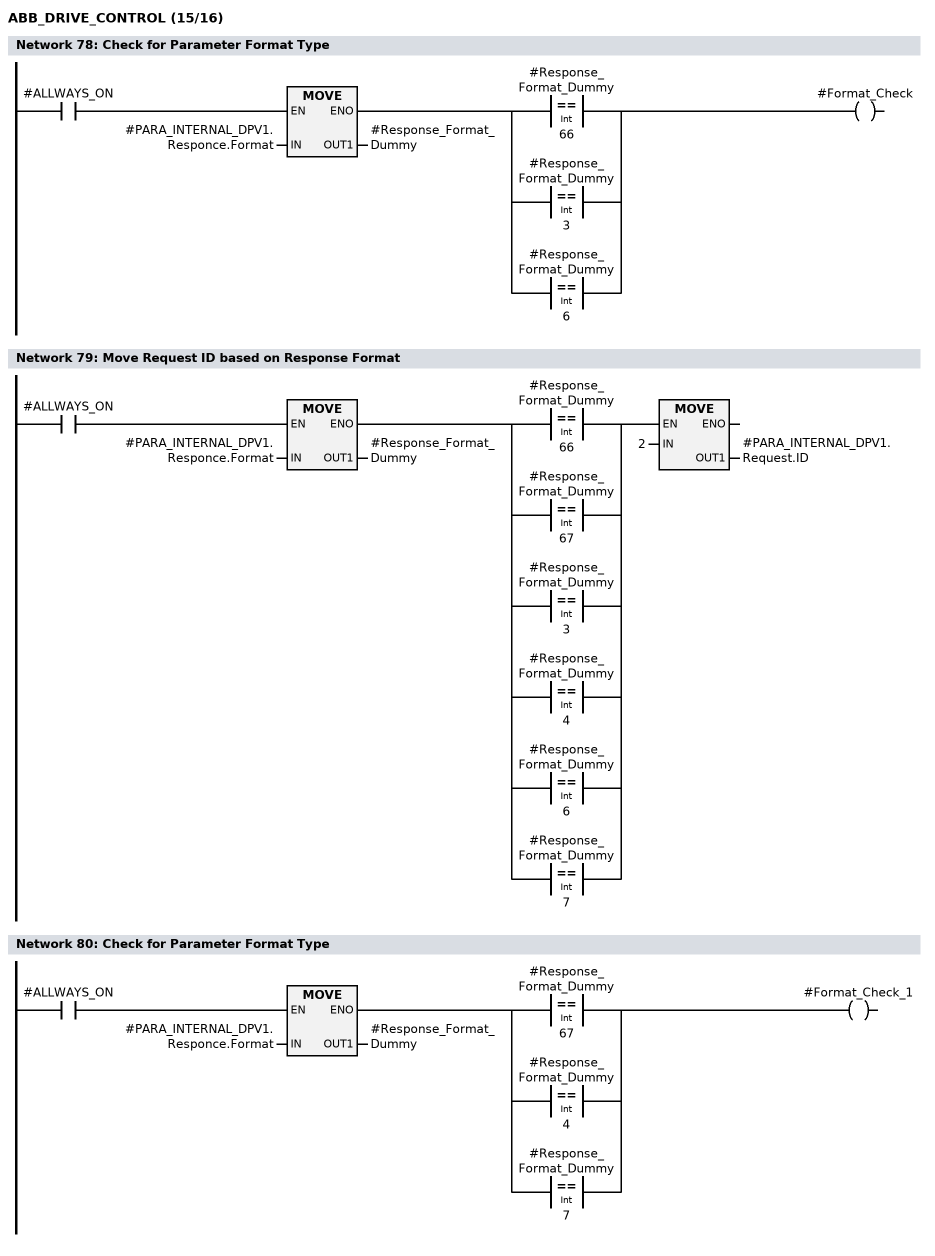
   RUNG wire#powerrail
      Contact( #ALLWAYS_ON )
      { S7_GenerateENO := "TRUE" } Move(in := #PARA_INTERNAL_DPV1.Responce.Format, out1 => #Response_Format_Dummy)
      wire#w1
      { S7_Templates := "SrcType := Int" } EQ_Contact(in1 := #Response_Format_Dummy, in2 := 66)
      wire#w2
      Coil( #Format_Check )
   END_RUNG
   RUNG wire#w1
      { S7_Templates := "SrcType := Int" } EQ_Contact(in1 := #Response_Format_Dummy, in2 := 3)
   END_RUNG wire#w2
   RUNG wire#w1
      { S7_Templates := "SrcType := Int" } EQ_Contact(in1 := #Response_Format_Dummy, in2 := 6)
   END_RUNG wire#w2
   // the same network as SCL:
   // ENO of a box is taken as its EN; it also drops when the box reports an error
   IF #ALLWAYS_ON THEN #Response_Format_Dummy := #PARA_INTERNAL_DPV1.Responce.Format; END_IF;
   #Format_Check := #ALLWAYS_ON AND ((#Response_Format_Dummy = 66) OR (#Response_Format_Dummy = 3) OR (#Response_Format_Dummy = 6));
END_REGION

REGION Network 79: Move Request ID based on Response Format
   RUNG wire#powerrail
      Contact( #ALLWAYS_ON )
      { S7_GenerateENO := "TRUE" } Move(in := #PARA_INTERNAL_DPV1.Responce.Format, out1 => #Response_Format_Dummy)
      wire#w1
      { S7_Templates := "SrcType := Int" } EQ_Contact(in1 := #Response_Format_Dummy, in2 := 66)
      wire#w2
      { S7_GenerateENO := "TRUE" } Move(in := 2, out1 => #PARA_INTERNAL_DPV1.Request.ID)
   END_RUNG
   RUNG wire#w1
      { S7_Templates := "SrcType := Int" } EQ_Contact(in1 := #Response_Format_Dummy, in2 := 67)
   END_RUNG wire#w2
   RUNG wire#w1
      { S7_Templates := "SrcType := Int" } EQ_Contact(in1 := #Response_Format_Dummy, in2 := 3)
   END_RUNG wire#w2
   RUNG wire#w1
      { S7_Templates := "SrcType := Int" } EQ_Contact(in1 := #Response_Format_Dummy, in2 := 4)
   END_RUNG wire#w2
   RUNG wire#w1
      { S7_Templates := "SrcType := Int" } EQ_Contact(in1 := #Response_Format_Dummy, in2 := 6)
   END_RUNG wire#w2
   RUNG wire#w1
      { S7_Templates := "SrcType := Int" } EQ_Contact(in1 := #Response_Format_Dummy, in2 := 7)
   END_RUNG wire#w2
   // the same network as SCL:
   // ENO of a box is taken as its EN; it also drops when the box reports an error
   IF #ALLWAYS_ON THEN #Response_Format_Dummy := #PARA_INTERNAL_DPV1.Responce.Format; END_IF;
   IF #ALLWAYS_ON AND ((#Response_Format_Dummy = 66) OR (#Response_Format_Dummy = 67) OR (#Response_Format_Dummy = 3) OR (#Response_Format_Dummy = 4) OR (#Response_Format_Dummy = 6) OR (#Response_Format_Dummy = 7)) THEN
       #PARA_INTERNAL_DPV1.Request.ID := 2;
   END_IF;
END_REGION

